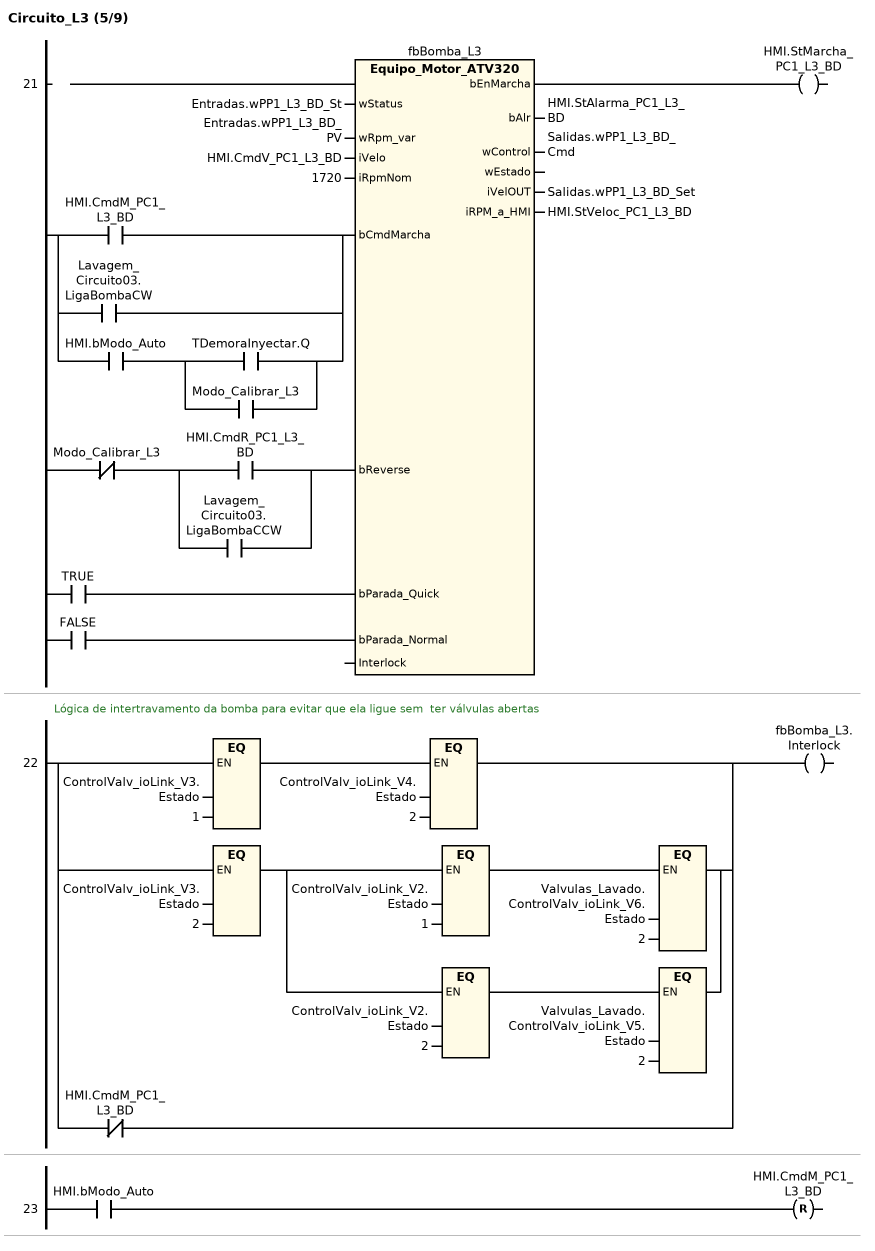
// NETWORK 21
fbBomba_L3(
    wStatus := Entradas.wPP1_L3_BD_St,
    wRpm_var := Entradas.wPP1_L3_BD_PV,
    iVelo := HMI.CmdV_PC1_L3_BD,
    iRpmNom := 1720,
    bCmdMarcha := HMI.CmdM_PC1_L3_BD OR Lavagem_Circuito03.LigaBombaCW OR HMI.bModo_Auto AND (TDemoraInyectar.Q OR Modo_Calibrar_L3),
    bReverse := NOT Modo_Calibrar_L3 AND (HMI.CmdR_PC1_L3_BD OR Lavagem_Circuito03.LigaBombaCCW),
    bParada_Quick := TRUE,
    bParada_Normal := FALSE,
    bAlr => HMI.StAlarma_PC1_L3_BD,
    wControl => Salidas.wPP1_L3_BD_Cmd,
    iVelOUT => Salidas.wPP1_L3_BD_Set,
    iRPM_a_HMI => HMI.StVeloc_PC1_L3_BD); // Equipo_Motor_ATV320
HMI.StMarcha_PC1_L3_BD := fbBomba_L3.bEnMarcha;

// NETWORK 22
// Lógica de intertravamento da bomba para evitar que ela ligue sem  ter válvulas abertas
_w6 := NOT HMI.CmdM_PC1_L3_BD;
IF NOT _w6 THEN
    _w7 := ControlValv_ioLink_V3.Estado = 2;
    _w6 := ControlValv_ioLink_V3.Estado = 1 AND ControlValv_ioLink_V4.Estado = 2 OR (_w7 AND ControlValv_ioLink_V2.Estado = 1 AND Valvulas_Lavado.ControlValv_ioLink_V6.Estado = 2 OR _w7 AND ControlValv_ioLink_V2.Estado = 2 AND Valvulas_Lavado.ControlValv_ioLink_V5.Estado = 2);
END_IF
fbBomba_L3.Interlock := _w6;

// NETWORK 23
HMI.CmdM_PC1_L3_BD R= HMI.bModo_Auto;

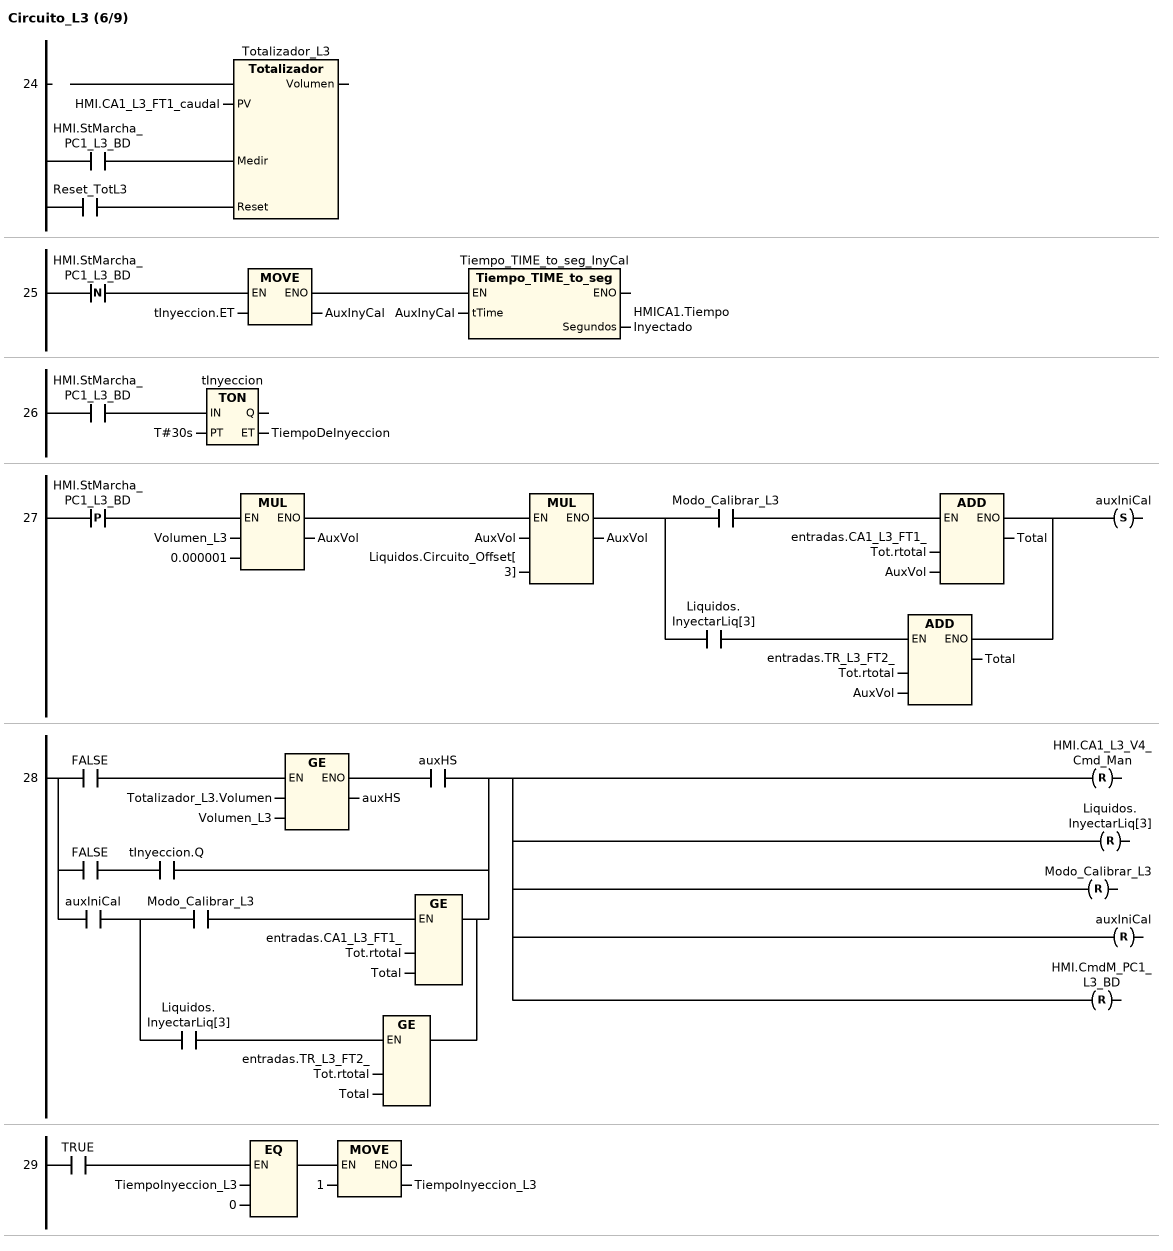
// NETWORK 24
Totalizador_L3(PV := HMI.CA1_L3_FT1_caudal, Medir := HMI.StMarcha_PC1_L3_BD, Reset := Reset_TotL3); // Totalizador

// NETWORK 25
_ft1(CLK := HMI.StMarcha_PC1_L3_BD);
_w8 := _ft1.Q;
IF _w8 THEN AuxInyCal := tInyeccion.ET; END_IF
IF _w8 THEN
    Tiempo_TIME_to_seg_InyCal(tTime := AuxInyCal, Segundos => HMICA1.TiempoInyectado); // Tiempo_TIME_to_seg
END_IF

// NETWORK 26
tInyeccion(IN := HMI.StMarcha_PC1_L3_BD, PT := T#30s, ET => TiempoDeInyeccion); // TON

// NETWORK 27
_rt1(CLK := HMI.StMarcha_PC1_L3_BD);
_w9 := _rt1.Q;
IF _w9 THEN AuxVol := Volumen_L3 * 0.000001; END_IF
IF _w9 THEN AuxVol := AuxVol * Liquidos.Circuito_Offset[3]; END_IF
IF _w9 AND Modo_Calibrar_L3 THEN Total := entradas.CA1_L3_FT1_Tot.rtotal + AuxVol; END_IF
IF _w9 AND Liquidos.InyectarLiq[3] THEN Total := entradas.TR_L3_FT2_Tot.rtotal + AuxVol; END_IF
auxIniCal S= _w9 AND Modo_Calibrar_L3 OR _w9 AND Liquidos.InyectarLiq[3];

// NETWORK 28
IF FALSE THEN auxHS := Totalizador_L3.Volumen >= Volumen_L3; END_IF
_w10 := FALSE AND auxHS OR FALSE AND tInyeccion.Q OR (auxIniCal AND Modo_Calibrar_L3 AND entradas.CA1_L3_FT1_Tot.rtotal >= Total OR auxIniCal AND Liquidos.InyectarLiq[3] AND entradas.TR_L3_FT2_Tot.rtotal >= Total);
HMI.CA1_L3_V4_Cmd_Man R= _w10;
Liquidos.InyectarLiq[3] R= _w10;
Modo_Calibrar_L3 R= _w10;
auxIniCal R= _w10;
HMI.CmdM_PC1_L3_BD R= _w10;

// NETWORK 29
IF TiempoInyeccion_L3 = 0 THEN TiempoInyeccion_L3 := 1; END_IF

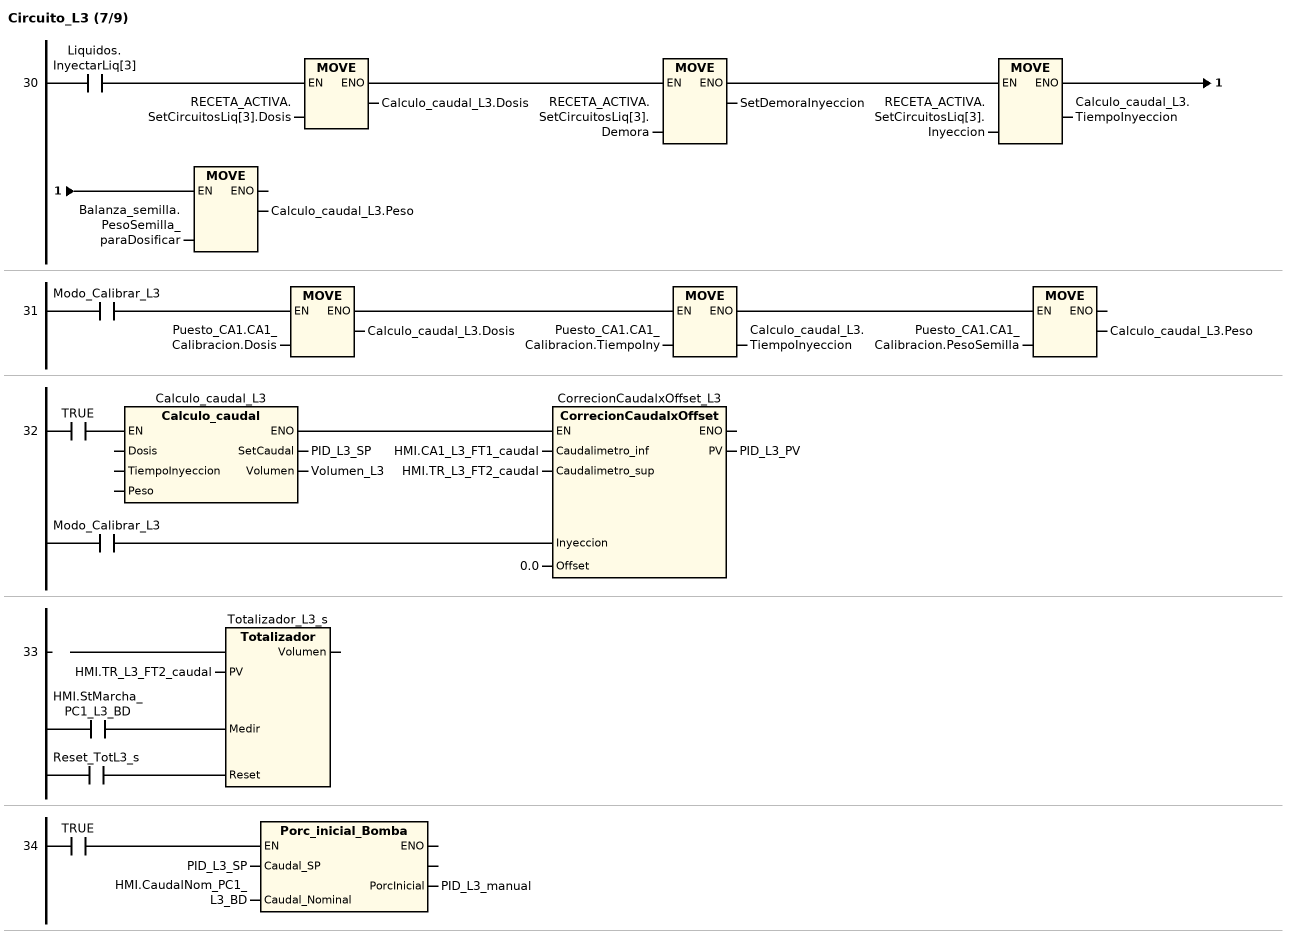
// NETWORK 30
_w11 := Liquidos.InyectarLiq[3];
IF _w11 THEN Calculo_caudal_L3.Dosis := RECETA_ACTIVA.SetCircuitosLiq[3].Dosis; END_IF
IF _w11 THEN SetDemoraInyeccion := RECETA_ACTIVA.SetCircuitosLiq[3].Demora; END_IF
IF _w11 THEN Calculo_caudal_L3.TiempoInyeccion := RECETA_ACTIVA.SetCircuitosLiq[3].Inyeccion; END_IF
IF _w11 THEN Calculo_caudal_L3.Peso := Balanza_semilla.PesoSemilla_paraDosificar; END_IF

// NETWORK 31
_w12 := Modo_Calibrar_L3;
IF _w12 THEN Calculo_caudal_L3.Dosis := Puesto_CA1.CA1_Calibracion.Dosis; END_IF
IF _w12 THEN Calculo_caudal_L3.TiempoInyeccion := Puesto_CA1.CA1_Calibracion.TiempoIny; END_IF
IF _w12 THEN Calculo_caudal_L3.Peso := Puesto_CA1.CA1_Calibracion.PesoSemilla; END_IF

// NETWORK 32
Calculo_caudal_L3(SetCaudal => PID_L3_SP, Volumen => Volumen_L3); // Calculo_caudal
CorrecionCaudalxOffset_L3(
    Caudalimetro_inf := HMI.CA1_L3_FT1_caudal,
    Caudalimetro_sup := HMI.TR_L3_FT2_caudal,
    Inyeccion := Modo_Calibrar_L3,
    Offset := 0.0,
    PV => PID_L3_PV); // CorrecionCaudalxOffset

// NETWORK 33
Totalizador_L3_s(PV := HMI.TR_L3_FT2_caudal, Medir := HMI.StMarcha_PC1_L3_BD, Reset := Reset_TotL3_s); // Totalizador

// NETWORK 34
Porc_inicial_Bomba(Caudal_SP := PID_L3_SP, Caudal_Nominal := HMI.CaudalNom_PC1_L3_BD, PorcInicial => PID_L3_manual);

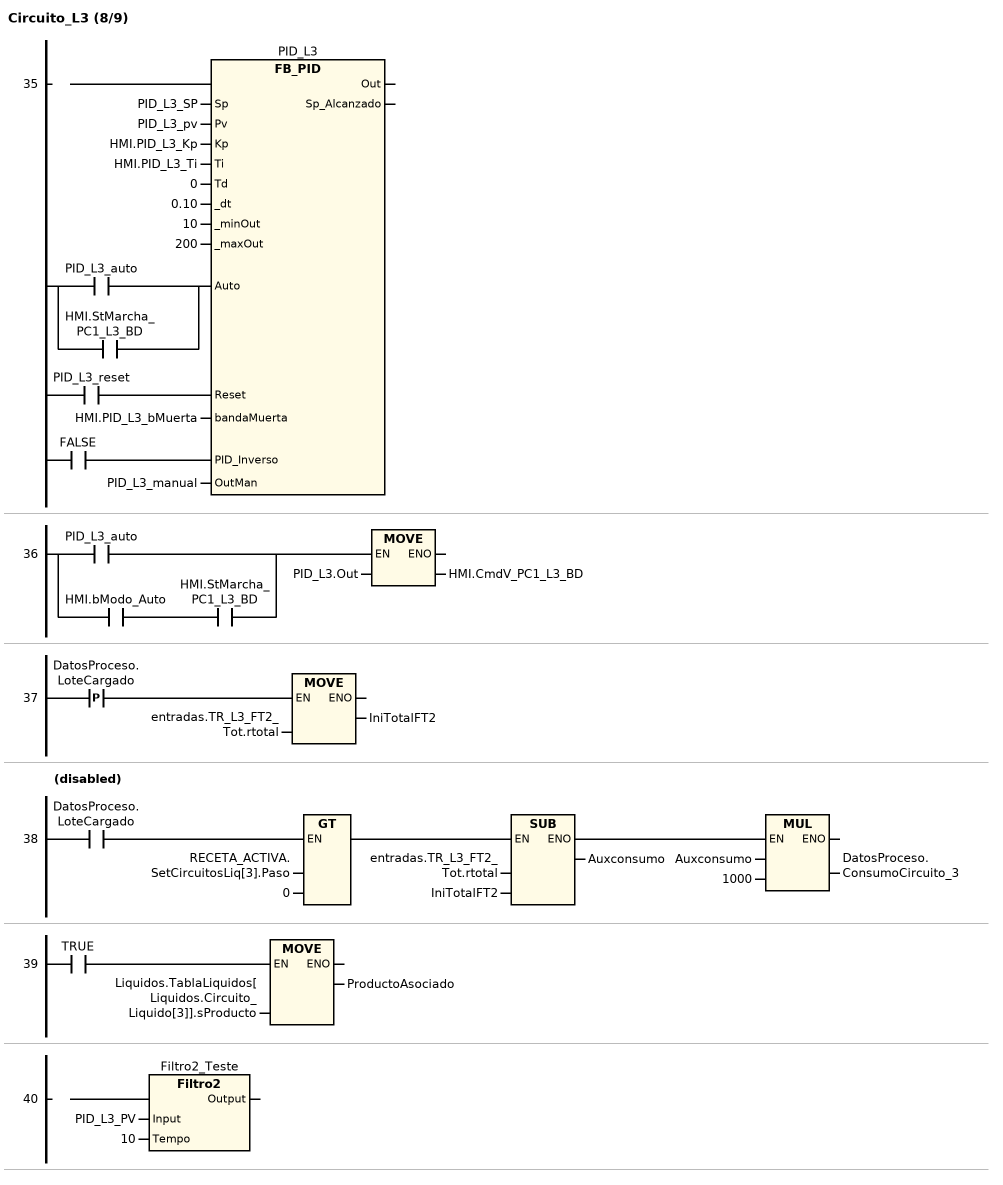
// NETWORK 35
PID_L3(
    Sp := PID_L3_SP,
    Pv := PID_L3_pv,
    Kp := HMI.PID_L3_Kp,
    Ti := HMI.PID_L3_Ti,
    Td := 0,
    _dt := 0.10,
    _minOut := 10,
    _maxOut := 200,
    Auto := PID_L3_auto OR HMI.StMarcha_PC1_L3_BD,
    Reset := PID_L3_reset,
    bandaMuerta := HMI.PID_L3_bMuerta,
    PID_Inverso := FALSE,
    OutMan := PID_L3_manual); // FB_PID

// NETWORK 36
IF PID_L3_auto OR HMI.bModo_Auto AND HMI.StMarcha_PC1_L3_BD THEN HMI.CmdV_PC1_L3_BD := PID_L3.Out; END_IF

// NETWORK 37
_rt2(CLK := DatosProceso.LoteCargado);
IF _rt2.Q THEN IniTotalFT2 := entradas.TR_L3_FT2_Tot.rtotal; END_IF

// NETWORK 38 (disabled)
// _w13 := DatosProceso.LoteCargado AND RECETA_ACTIVA.SetCircuitosLiq[3].Paso > 0;
// IF _w13 THEN Auxconsumo := entradas.TR_L3_FT2_Tot.rtotal - IniTotalFT2; END_IF
// IF _w13 THEN DatosProceso.ConsumoCircuito_3 := Auxconsumo * 1000; END_IF

// NETWORK 39
ProductoAsociado := Liquidos.TablaLiquidos[Liquidos.Circuito_Liquido[3]].sProducto;

// NETWORK 40
Filtro2_Teste(Input := PID_L3_PV, Tempo := 10); // Filtro2

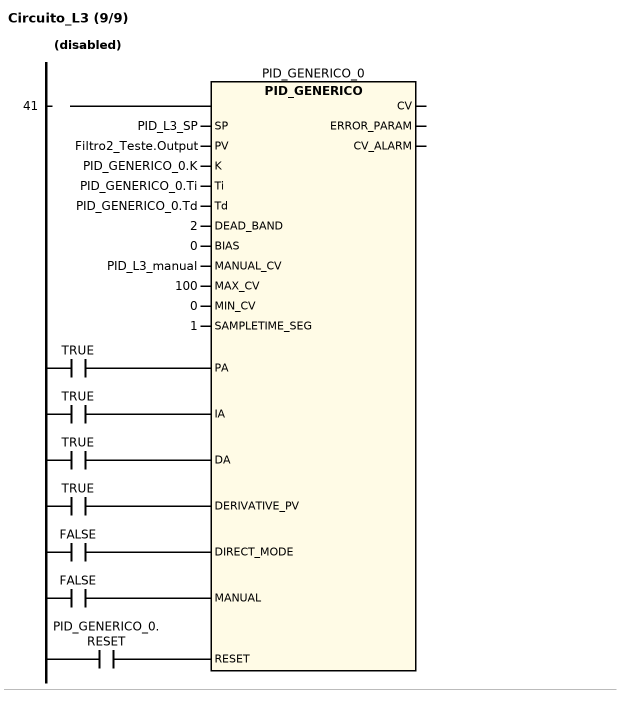
// NETWORK 41 (disabled)
// PID_GENERICO_0(
//     SP := PID_L3_SP,
//     PV := Filtro2_Teste.Output,
//     K := PID_GENERICO_0.K,
//     Ti := PID_GENERICO_0.Ti,
//     Td := PID_GENERICO_0.Td,
//     DEAD_BAND := 2,
//     BIAS := 0,
//     MANUAL_CV := PID_L3_manual,
//     MAX_CV := 100,
//     MIN_CV := 0,
//     SAMPLETIME_SEG := 1,
//     PA := TRUE,
//     IA := TRUE,
//     DA := TRUE,
//     DERIVATIVE_PV := TRUE,
//     DIRECT_MODE := FALSE,
//     MANUAL := FALSE,
//     RESET := PID_GENERICO_0.RESET); // PID_GENERICO

END_PROGRAM

// ---- POUs/TestesPID/PID_GENERICO.TcPOU
FUNCTION_BLOCK PID_GENERICO

VAR_INPUT
	SP: REAL; //SETPOINT
	PV: REAL; //VARIAVEL DE PROCESSO (ENTRADA)
	K: REAL; //GANHO PROPORCIONAL
	Ti: REAL; //GANHO INTEGRAL (TEMPO INTEGRAL)
	Td: REAL; //GANHO REAL (TEMPO DERIVATIVO)
	DEAD_BAND: REAL; //BANDA MORTA
	BIAS: REAL; //BIAS - VALOR SOMANDO A SAIDA DO CONTROLADOR
	MANUAL_CV: REAL; //VALOR DA SAIDA QUANDO O MANUAL ESTIVER HABILITADO
	MAX_CV: REAL; //VALOR MAXIMO DA SAIDA
	MIN_CV: REAL; //VALOR MINIMO DA SAIDA
	SAMPLETIME_SEG:REAL; //TEMPO DE ATUALIZAÇÃO DA TASK
	PA: BOOL; //HABILITA FATOR PROPORCIONAL
	IA: BOOL; //HABILITA FATOR INTEGRAL
	DA: BOOL; //HABILITA FATOR DERIVATIVO
	DERIVATIVE_PV: BOOL; //ADICIONAR FATOR DERIVATIVO A VARIAVEL DE PROCESSO
	DIRECT_MODE: BOOL; //MODO DIRETO OU REVERSO
	MANUAL: BOOL; //HABILITA MODO MANUAL
	RESET: BOOL; //RESET DO BLOCO
END_VAR
VAR_OUTPUT
	CV: INT; //VARIAVEL DE CONTROLE (SAIDA)
	ERROR_PARAM: BOOL; //ERRO DE PARAMETRO
	CV_ALARM: BOOL; //ALARME DE LIMITES DA SAIDA ATINGIDO (SATURAÇÃO)
END_VAR
VAR
	RealCV : REAL := 0;
	RealTimeCycle: ARRAY [0..2] OF REAL := [0,0,0];
	RealSystemError: ARRAY [0..3] OF REAL := [0,0,0,0];
	RealProcessVariable: ARRAY [0..3] OF REAL := [0,0,0,0];
	RealProportionalAction: REAL := 0;
	RealIntegralAction: REAL := 0;
	RealDerivativeAction: REAL := 0;
	RealIntegralLastAction: REAL := 0;
	DwCurrentReferenceCycle: DWORD;
	DwLastReferenceCycle:DWORD := 0;
	BoolFirstCycle: BOOL := TRUE;
END_VAR


(*###################################################################################                                                     
##  									                                      								                                      
##	Function Block Name: PID_FB                                                                                                                                  
##  									                                      								                                      
##  Version: 1.00                                                                                                                                                                 
##  									                                      								                                      
##                                                                                                
##  									                                      								                                      
##  Software Description: The PID function block implements the proportional, integral and derivative          
##  control algorithm. Using a process variable (PV) and a setpoint (SP) the function computes the              
##  control variable (CV) for the process under control. This value is calculated periodically, and 
##  takes into consideration the proportional, integral and derivative configured factors. This is a ISA 
##  PID control algorithm in which the proportional gain is the controller gain, that is applied to the 
##  controller error as well as it's integral and derivative terms.
##
###################################################################################*)




(* ----------------------------------------------------------  RESET TREATMENT-------------------------------------------------------*)
IF(RESET = TRUE)
THEN
		RealSystemError[0] := 0;
		RealSystemError[1] := 0;
		RealSystemError[2] := 0;
		RealSystemError[3] := 0;
		RealProcessVariable[0] := 0;
		RealProcessVariable[1] := 0;
		RealProcessVariable[2] := 0;
		RealProcessVariable[3] := 0;
		RealTimeCycle[0] := 0;
		RealTimeCycle[1] := 0;
		RealTimeCycle[2] := 0;
		RealIntegralLastAction := 0;
		BoolFirstCycle:= TRUE;

		(* Reset the output variables*)
		ERROR_PARAM := FALSE;
		CV_ALARM := FALSE;
		CV := 0;
		RETURN;
END_IF;
(*############################## END OF RESET TREATMENT ############################*)


(*------------------------------------------------------- PARAMETERS TEST -----------------------------------------------------------*)
IF(K<=0 OR Ti<=0 OR Td<0 OR MAX_CV<MIN_CV OR MAX_CV>32767 OR MIN_CV<-32768)
THEN
		RealSystemError[0] := 0;
		RealSystemError[1] := 0;
		RealSystemError[2] := 0;
		RealSystemError[3] := 0;
		RealProcessVariable[0] := 0;
		RealProcessVariable[1] := 0;
		RealProcessVariable[2] := 0;
		RealProcessVariable[3] := 0;
		RealTimeCycle[0] := 0;
		RealTimeCycle[1] := 0;
		RealTimeCycle[2] := 0;
		RealIntegralLastAction := 0;
		BoolFirstCycle:= TRUE;
		CV_ALARM := FALSE;
		ERROR_PARAM:= TRUE;
		CV:= 0;
		RETURN;
ELSE
		ERROR_PARAM:= FALSE;
END_IF;

(*############################## END PARAMETERS TEST ###############################*)

(*------------------ KEEPS A LOG OF THE LAST FOUR ERRORS  AND PROCESS VARIABLES ----------------------*)

RealSystemError[3] := RealSystemError[2];
RealSystemError[2] := RealSystemError[1];
RealSystemError[1] := RealSystemError[0];

RealProcessVariable[3] := RealProcessVariable[2];
RealProcessVariable[2] := RealProcessVariable[1];
RealProcessVariable[1] := RealProcessVariable[0];

IF(DIRECT_MODE = TRUE)
THEN	RealSystemError[0]:=PV - SP;
		RealProcessVariable[0 ]:= -PV;

ELSE	RealSystemError[0]:=SP -PV;
		RealProcessVariable[0 ]:= PV;
END_IF;


(*  Applys the dead band over the system error *)
IF(ABS(RealSystemError[0]) <= ABS(DEAD_BAND))
THEN	RealSystemError[0]:= 0;
END_IF;

(*################################ END OF ERRORS AND PV LOG ############################*)


(*------------------------------------------------------ TIME BASE DEFINITION ----------------------------------------------------------*)


IF(BoolFirstCycle = FALSE)
THEN
		RealTimeCycle[2] := SAMPLETIME_SEG;
		RealTimeCycle[1] := SAMPLETIME_SEG;
		RealTimeCycle[0]:= SAMPLETIME_SEG;

		IF(RealTimeCycle[0] = 0)		(* If the current cycle is less than 1 ms it is forced do 1 ms *)
		THEN	RealTimeCycle[0] := 0.001;
		END_IF;
ELSE
		BoolFirstCycle := FALSE;
		RETURN;
END_IF;
(*############################# END OF TIME BASE DEFINITION  ############################*)


(* -----------------------------------------------------  PROPORTIONAL ACTION -----------------------------------------------------*)
 IF (PA = TRUE)
THEN
		(* The proportional action is only the current error *)
		(* Remind that "K" is the controller gain and it will be applied to the sum of proportional integral and derivative actions *)
		RealProportionalAction := RealSystemError[0];
ELSE
		(* If the proportional action is not desirable its value would be zero *)
		RealProportionalAction := 0;
END_IF;
(*############################ END OF PROPORTIONAL ACTION #############################*)


(* ---------------------------------------------------------  INTEGRAL ACTION ---------------------------------------------------------*)
IF( IA = TRUE AND MANUAL = FALSE)
THEN
		(* It keeps the last egral Action because it must be used when the controled variable reaches its limits *)
		RealIntegralLastAction := RealIntegralAction;

		(* The integral action is the amount  obtained from the current system error multiplied by the sample time and
		    divided by  the the programmed integral time*)

		(* Remind that "K" is the controller gain and it will be applied to the sum of proportional integral and derivative actions *)
		RealIntegralAction := RealIntegralLastAction + RealSystemError[0] * RealTimeCycle[0] / Ti;

		(* Limits the integral action in 10 times the maximum output *)
		IF(RealIntegralAction > 327670)
		THEN	RealIntegralAction := 327670;
		END_IF;

		IF(RealIntegralAction < -327670)
		THEN	RealIntegralAction := -327670;
		END_IF;
ELSE
		(* If the Integral action is not desirable its value will be zero *)
		RealIntegralAction:= 0;
END_IF;
(*################################ END OF INTEGRAL ACTION ##############################*)


(* --------------------------------------------------------  DERIVATIVE ACTION --------------------------------------------------------*)
IF (DA = TRUE)
THEN
		(* The derivative action is the variation of de error during 3 cycles multiplied by the programmed derivative time*)
		(* Remind that "K" is the controller gain and it will be applied to the sum of proportional integral and derivative actions *)
		IF(DERIVATIVE_PV = TRUE)
		THEN	RealDerivativeAction:=  Td * (RealProcessVariable[3] - RealProcessVariable[0]) / (RealTimeCycle[0] + RealTimeCycle[1] + RealTimeCycle[2]);
		ELSE	RealDerivativeAction:=  Td * (RealSystemError[0] - RealSystemError[3]) / (RealTimeCycle[0] + RealTimeCycle[1] + RealTimeCycle[2]);
		END_IF;

		(* Limits the derivative action in 10 times the maximum output *)
		IF(RealDerivativeAction > 327670)
		THEN	RealDerivativeAction := 327670;
		END_IF;

		IF(RealDerivativeAction < -327670)
		THEN	RealDerivativeAction := -327670;
		END_IF;
ELSE
		(* If the derivative action is not desirable its value will be zero *)
		RealDerivativeAction:=0;
END_IF;
(*###############################  END OF DERIVATIVE ACTION ############################*)


(*-------------------------------------------- TESTS MANUAL OR AUTOMATIC MODE -----------------------------------------*)
IF(MANUAL = FALSE)
THEN
		(* in automatic mode the control variable is the sum of  the three actions  *)
		RealCV := K*(RealProportionalAction + RealIntegralAction + RealDerivativeAction) + BIAS;

		(* limits the output in the maximum programmed *)
		IF(RealCV > MAX_CV)
		THEN	CV := REAL_TO_INT(MAX_CV);
				CV_ALARM := TRUE;    (*indicates that the ouput reaches the limit*)
				(* keeps the current Integral Action only if the system error is negative *)
				IF(RealSystemError[0] > 0)
				THEN	RealIntegralAction := RealIntegralLastAction;
				END_IF;

		(* limits the output in the minimum programmed *)
		ELSE	IF(RealCV <  MIN_CV)
				THEN	CV := REAL_TO_INT(MIN_CV);
						CV_ALARM := TRUE;     (*indicates that the ouput reaches the limit*)
						(* keeps the current Integral Action only if the system error is positive *)
						IF(RealSystemError[0] < 0)
						THEN	RealIntegralAction := RealIntegralLastAction;
						END_IF;
				ELSE	CV := REAL_TO_INT(RealCV);
						CV_ALARM := FALSE;    (*indicates that the ouput is between the limits*)
				END_IF;
		END_IF;
ELSE
		(*In  manual mode the manual value is copied to the control variable .
		The stored integral action will be the difference between the CV_MANUAL and the Proportional, Derivative Actions
		and the programmed FF_Bias. *)

		(* If the Manual CV is configured above or below to the limits the control variable alarm is set and the CV will be
                 forced to the closest limit*)

		IF(MANUAL_CV > MAX_CV)
		THEN	CV := REAL_TO_INT(MAX_CV);
				CV_ALARM := TRUE;
		ELSE
				IF(MANUAL_CV <MIN_CV)
			    	THEN	CV := REAL_TO_INT(MIN_CV);
						CV_ALARM := TRUE;

				ELSE	CV := REAL_TO_INT(MANUAL_CV);
						CV_ALARM := FALSE;

				END_IF;
		END_IF;

		(*This Integral Action will be used in case of switch to automatic mode to ensure a smooth transition. *)
		RealIntegralAction:= (INT_TO_REAL(CV) - BIAS) / K - RealProportionalAction - RealDerivativeAction;

END_IF;

(*###############################  END MANUAL / AUTOMATIC ############################*)

END_FUNCTION_BLOCK

// ---- POUs/Secuencias/Porc_inicial_Bomba.TcPOU
FUNCTION Porc_inicial_Bomba : BOOL
VAR_INPUT
	Caudal_SP:REAL;
	Caudal_Nominal:REAL;
END_VAR
VAR_OUTPUT
	PorcInicial:REAL;
END_VAR
VAR
END_VAR

IF Caudal_Nominal=0 THEN
	Caudal_Nominal:=1;
END_IF
PorcInicial:=(Caudal_SP/Caudal_Nominal)*100.0*1.0;

END_FUNCTION

// ---- POUs/Puesto_Calibracion_1/Circuito_L4.TcPOU
PROGRAM Circuito_L4
VAR_INPUT
	Modo_Calibrar_L4: BOOL;
END_VAR
	
VAR
		fbBomba_L4 :Equipo_Motor_ATV320;
		ControlValv_ioLink_V1:ControlValv_ioLink;
		ControlValv_ioLink_V2: ControlValv_ioLink;
		ControlValv_ioLink_V3: ControlValv_ioLink;
		ControlValv_ioLink_V4: ControlValv_ioLink;
		Falla_L4_V1:BOOL;
		Falla_L4_V2:BOOL;
		Falla_L4_V3:BOOL;
		Falla_L4_V4:BOOL;
	Balanza_PU1_WT4: Balanza;
		dHS:DINT;
		TOF_calibradoIBC: TOF;
		TDemoraInyectar: TON;
		SetDemoraInyeccion: REAL;
	

	Volumen_L4: REAL;
	AuxVol: REAL;
	Total: REAL;
	auxIniCal: BOOL;
	Calculo_caudal_L4: Calculo_caudal;
	PID_L4_SP: REAL;
	PID_L4_PV: REAL;
	CorrecionCaudalxOffset_L4: CorrecionCaudalxOffset;
	tInyeccion: TON;
	PID_L4_manual: REAL;
	PID_L4: FB_PID;
	PID_L4_Kp: REAL := 0.1;
	PID_L4_Ti: REAL := 100;
	PID_L4_auto: BOOL;
	PID_L4_reset: BOOL;
	PID_L4_bMuerta: REAL := 5;
	Tiempo_seg_to_TIME_DemoraInyec: Tiempo_seg_to_TIME;
	AuxTDemoraInyec: TIME;
	Tiempo_TIME_to_seg_InyCal: Tiempo_TIME_to_seg;
	AuxInyCal:TIME;
	IniTotalFT2:REAL;
	Auxconsumo:REAL;
	ProductoAsociado: STRING;
	Lavagem_Circuito04: Lavagem;
	
END_VAR
VAR PERSISTENT
	UltimaCalibracao	:UDINT;	//Data e hora da ultima calibração
END_VAR
VAR // added by the converter: edge detectors and wires of the graphical bodies
    _w1, _w2, _w3, _w4, _w5, _w6, _w7, _w8, _w9, _w10, _w11, _w12, _w13 : BOOL;
    _ft1 : F_TRIG;
    _rt1, _rt2 : R_TRIG;
END_VAR

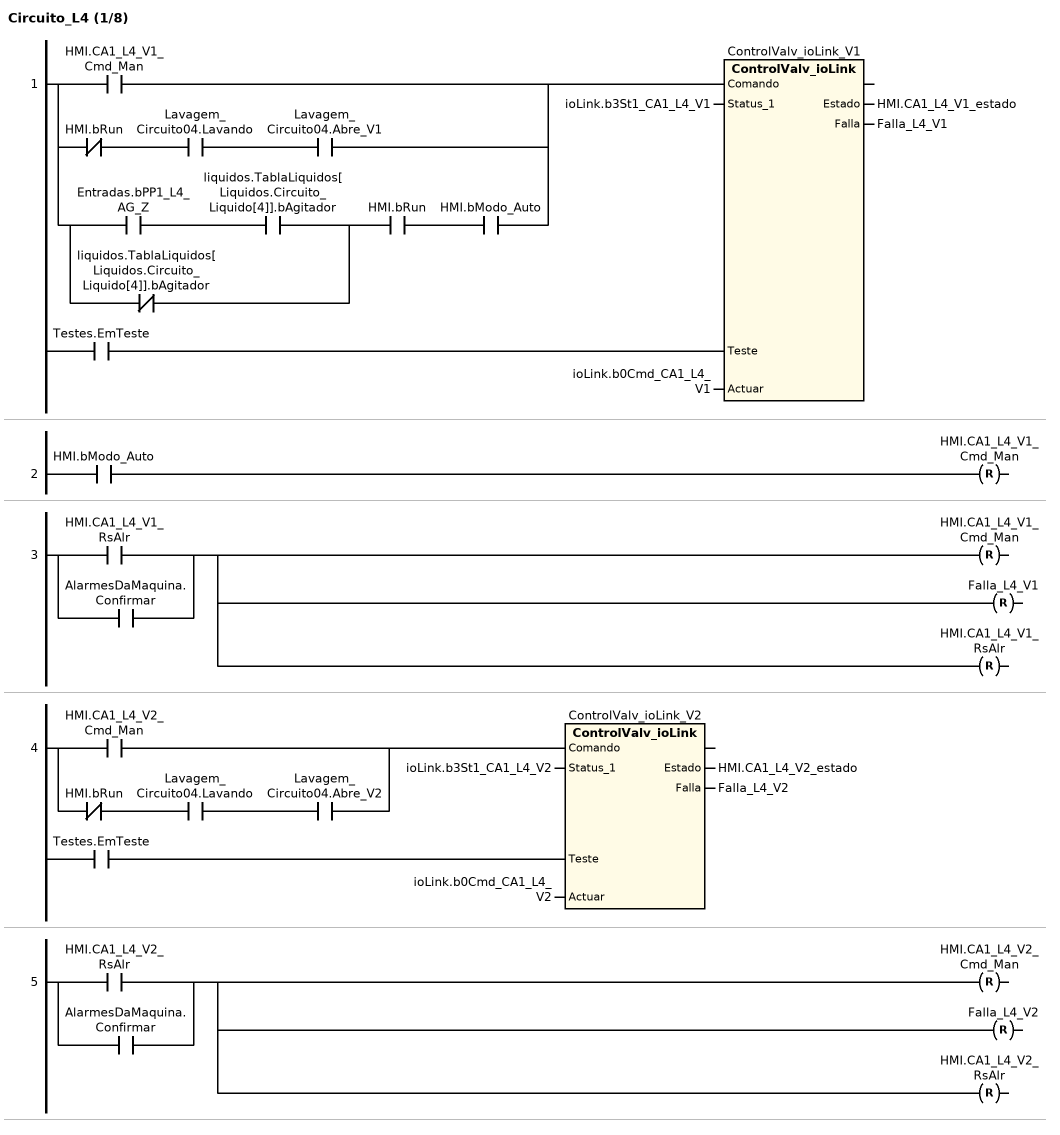
// NETWORK 1
ControlValv_ioLink_V1(
    Comando := HMI.CA1_L4_V1_Cmd_Man OR NOT HMI.bRun AND Lavagem_Circuito04.Lavando AND Lavagem_Circuito04.Abre_V1 OR (Entradas.bPP1_L4_AG_Z AND (liquidos.TablaLiquidos[Liquidos.Circuito_Liquido[4]].bAgitador) OR NOT (liquidos.TablaLiquidos[Liquidos.Circuito_Liquido[4]].bAgitador)) AND HMI.bRun AND HMI.bModo_Auto,
    Status_1 := ioLink.b3St1_CA1_L4_V1,
    Teste := Testes.EmTeste,
    Actuar := ioLink.b0Cmd_CA1_L4_V1,
    Estado => HMI.CA1_L4_V1_estado,
    Falla => Falla_L4_V1); // ControlValv_ioLink

// NETWORK 2
HMI.CA1_L4_V1_Cmd_Man R= HMI.bModo_Auto;

// NETWORK 3
_w1 := HMI.CA1_L4_V1_RsAlr OR AlarmesDaMaquina.Confirmar;
HMI.CA1_L4_V1_Cmd_Man R= _w1;
Falla_L4_V1 R= _w1;
HMI.CA1_L4_V1_RsAlr R= _w1;

// NETWORK 4
ControlValv_ioLink_V2(
    Comando := HMI.CA1_L4_V2_Cmd_Man OR NOT HMI.bRun AND Lavagem_Circuito04.Lavando AND Lavagem_Circuito04.Abre_V2,
    Status_1 := ioLink.b3St1_CA1_L4_V2,
    Teste := Testes.EmTeste,
    Actuar := ioLink.b0Cmd_CA1_L4_V2,
    Estado => HMI.CA1_L4_V2_estado,
    Falla => Falla_L4_V2); // ControlValv_ioLink

// NETWORK 5
_w2 := HMI.CA1_L4_V2_RsAlr OR AlarmesDaMaquina.Confirmar;
HMI.CA1_L4_V2_Cmd_Man R= _w2;
Falla_L4_V2 R= _w2;
HMI.CA1_L4_V2_RsAlr R= _w2;

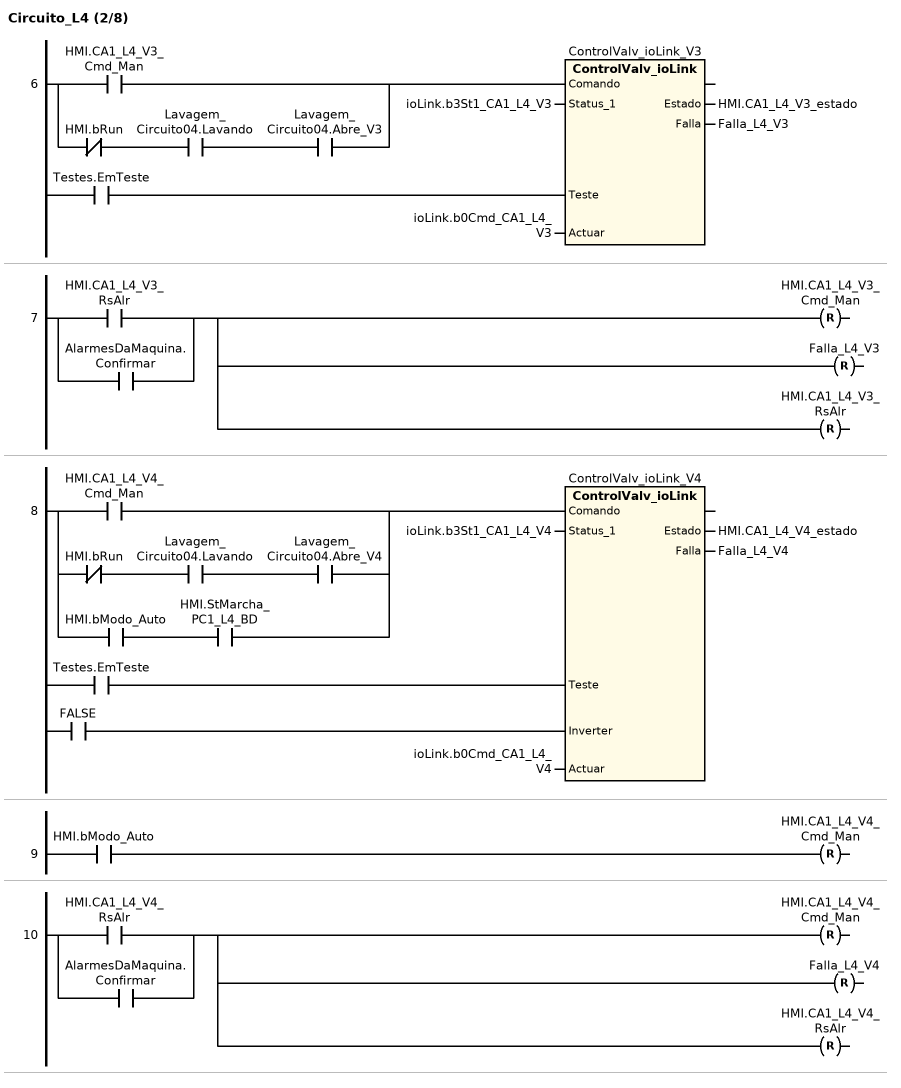
// NETWORK 6
ControlValv_ioLink_V3(
    Comando := HMI.CA1_L4_V3_Cmd_Man OR NOT HMI.bRun AND Lavagem_Circuito04.Lavando AND Lavagem_Circuito04.Abre_V3,
    Status_1 := ioLink.b3St1_CA1_L4_V3,
    Teste := Testes.EmTeste,
    Actuar := ioLink.b0Cmd_CA1_L4_V3,
    Estado => HMI.CA1_L4_V3_estado,
    Falla => Falla_L4_V3); // ControlValv_ioLink

// NETWORK 7
_w3 := HMI.CA1_L4_V3_RsAlr OR AlarmesDaMaquina.Confirmar;
HMI.CA1_L4_V3_Cmd_Man R= _w3;
Falla_L4_V3 R= _w3;
HMI.CA1_L4_V3_RsAlr R= _w3;

// NETWORK 8
ControlValv_ioLink_V4(
    Comando := HMI.CA1_L4_V4_Cmd_Man OR NOT HMI.bRun AND Lavagem_Circuito04.Lavando AND Lavagem_Circuito04.Abre_V4 OR HMI.bModo_Auto AND HMI.StMarcha_PC1_L4_BD,
    Status_1 := ioLink.b3St1_CA1_L4_V4,
    Teste := Testes.EmTeste,
    Inverter := FALSE,
    Actuar := ioLink.b0Cmd_CA1_L4_V4,
    Estado => HMI.CA1_L4_V4_estado,
    Falla => Falla_L4_V4); // ControlValv_ioLink

// NETWORK 9
HMI.CA1_L4_V4_Cmd_Man R= HMI.bModo_Auto;

// NETWORK 10
_w4 := HMI.CA1_L4_V4_RsAlr OR AlarmesDaMaquina.Confirmar;
HMI.CA1_L4_V4_Cmd_Man R= _w4;
Falla_L4_V4 R= _w4;
HMI.CA1_L4_V4_RsAlr R= _w4;

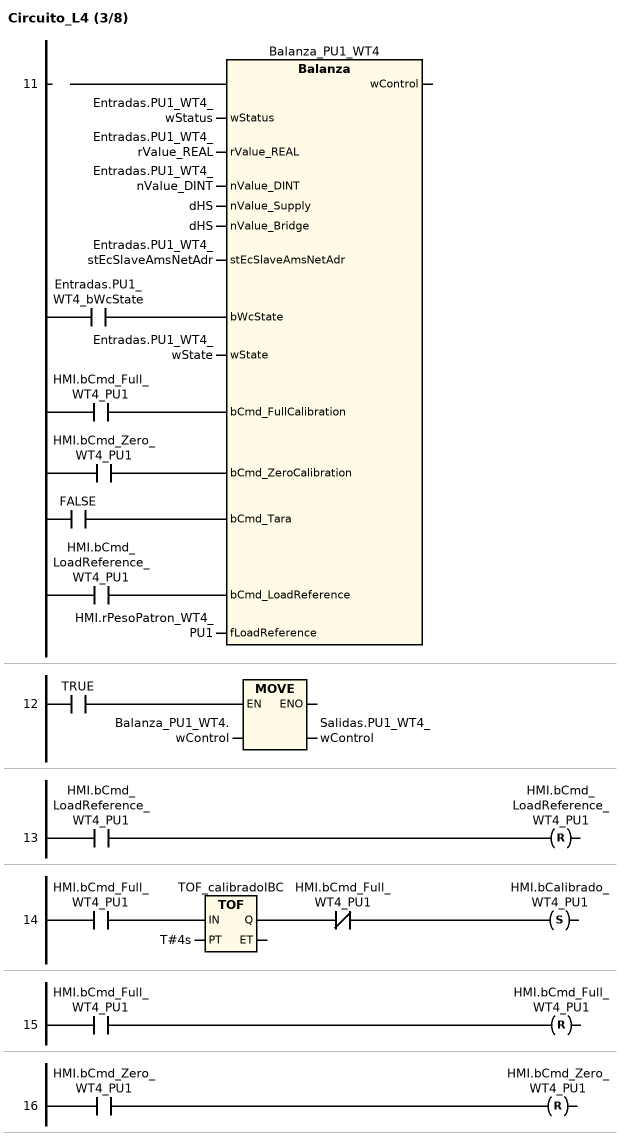
// NETWORK 11
Balanza_PU1_WT4(
    wStatus := Entradas.PU1_WT4_wStatus,
    rValue_REAL := Entradas.PU1_WT4_rValue_REAL,
    nValue_DINT := Entradas.PU1_WT4_nValue_DINT,
    nValue_Supply := dHS,
    nValue_Bridge := dHS,
    stEcSlaveAmsNetAdr := Entradas.PU1_WT4_stEcSlaveAmsNetAdr,
    bWcState := Entradas.PU1_WT4_bWcState,
    wState := Entradas.PU1_WT4_wState,
    bCmd_FullCalibration := HMI.bCmd_Full_WT4_PU1,
    bCmd_ZeroCalibration := HMI.bCmd_Zero_WT4_PU1,
    bCmd_Tara := FALSE,
    bCmd_LoadReference := HMI.bCmd_LoadReference_WT4_PU1,
    fLoadReference := HMI.rPesoPatron_WT4_PU1); // Balanza

// NETWORK 12
Salidas.PU1_WT4_wControl := Balanza_PU1_WT4.wControl;

// NETWORK 13
HMI.bCmd_LoadReference_WT4_PU1 R= HMI.bCmd_LoadReference_WT4_PU1;

// NETWORK 14
TOF_calibradoIBC(IN := HMI.bCmd_Full_WT4_PU1, PT := T#4s); // TOF
HMI.bCalibrado_WT4_PU1 S= TOF_calibradoIBC.Q AND NOT HMI.bCmd_Full_WT4_PU1;

// NETWORK 15
HMI.bCmd_Full_WT4_PU1 R= HMI.bCmd_Full_WT4_PU1;

// NETWORK 16
HMI.bCmd_Zero_WT4_PU1 R= HMI.bCmd_Zero_WT4_PU1;

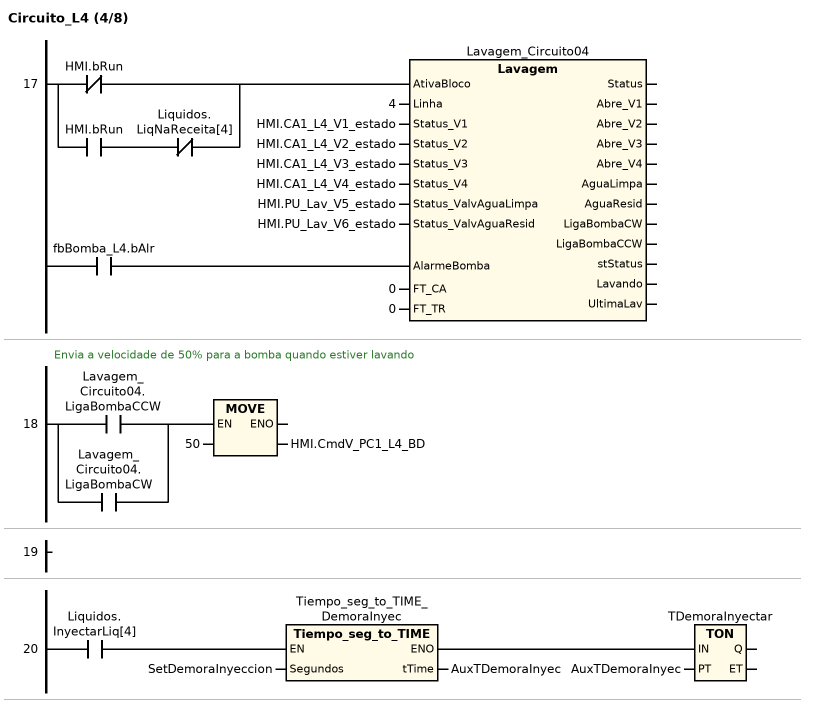
// NETWORK 17
Lavagem_Circuito04(
    AtivaBloco := NOT HMI.bRun OR HMI.bRun AND NOT Liquidos.LiqNaReceita[4],
    Linha := 4,
    Status_V1 := HMI.CA1_L4_V1_estado,
    Status_V2 := HMI.CA1_L4_V2_estado,
    Status_V3 := HMI.CA1_L4_V3_estado,
    Status_V4 := HMI.CA1_L4_V4_estado,
    Status_ValvAguaLimpa := HMI.PU_Lav_V5_estado,
    Status_ValvAguaResid := HMI.PU_Lav_V6_estado,
    AlarmeBomba := fbBomba_L4.bAlr,
    FT_CA := 0,
    FT_TR := 0); // Lavagem

// NETWORK 18
// Envia a velocidade de 50% para a bomba quando estiver lavando
IF Lavagem_Circuito04.LigaBombaCCW OR Lavagem_Circuito04.LigaBombaCW THEN HMI.CmdV_PC1_L4_BD := 50; END_IF

// NETWORK 19

// NETWORK 20
_w5 := Liquidos.InyectarLiq[4];
IF _w5 THEN
    Tiempo_seg_to_TIME_DemoraInyec(Segundos := SetDemoraInyeccion, tTime => AuxTDemoraInyec); // Tiempo_seg_to_TIME
END_IF
TDemoraInyectar(IN := _w5, PT := AuxTDemoraInyec); // TON

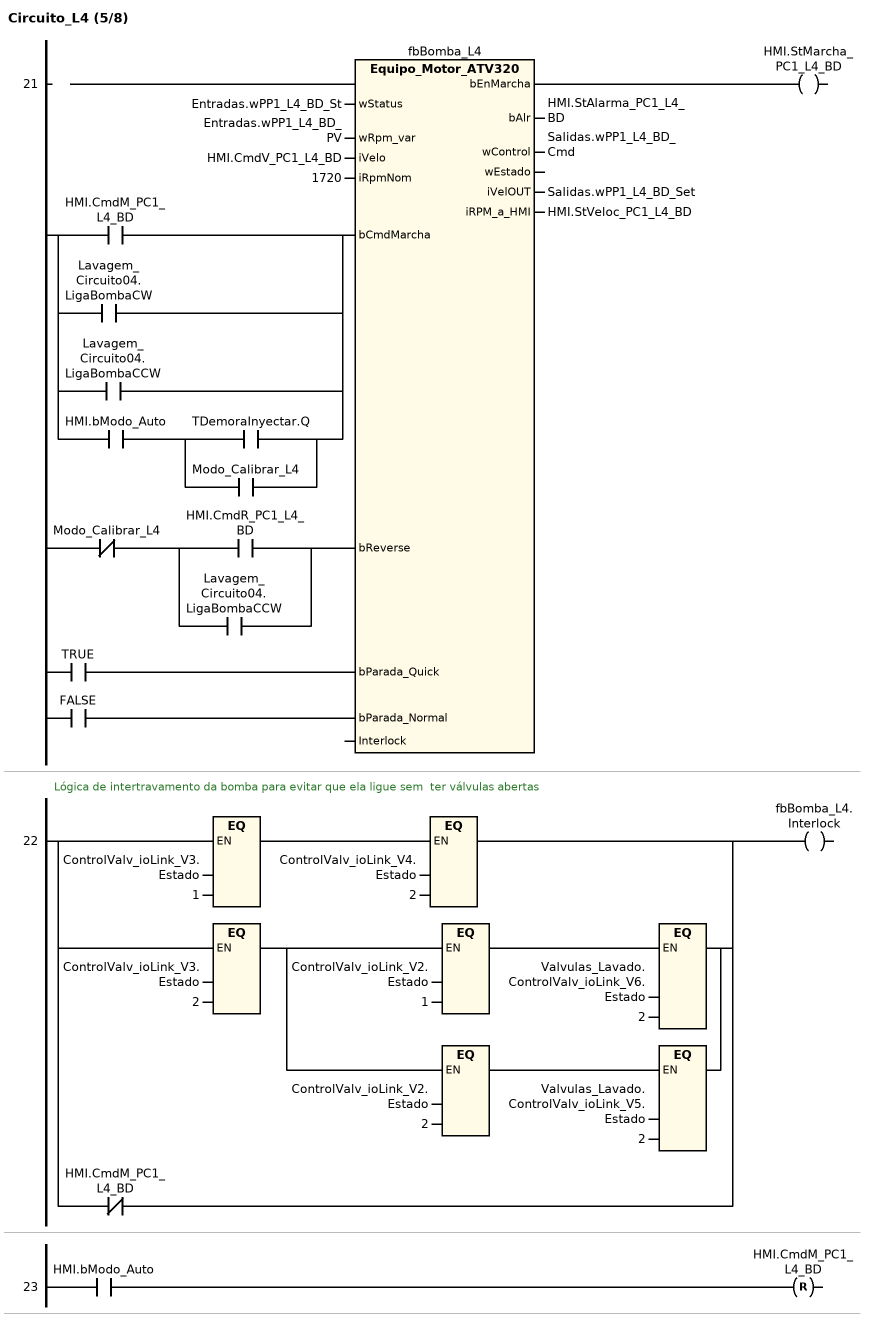
// NETWORK 21
fbBomba_L4(
    wStatus := Entradas.wPP1_L4_BD_St,
    wRpm_var := Entradas.wPP1_L4_BD_PV,
    iVelo := HMI.CmdV_PC1_L4_BD,
    iRpmNom := 1720,
    bCmdMarcha := HMI.CmdM_PC1_L4_BD OR Lavagem_Circuito04.LigaBombaCW OR Lavagem_Circuito04.LigaBombaCCW OR HMI.bModo_Auto AND (TDemoraInyectar.Q OR Modo_Calibrar_L4),
    bReverse := NOT Modo_Calibrar_L4 AND (HMI.CmdR_PC1_L4_BD OR Lavagem_Circuito04.LigaBombaCCW),
    bParada_Quick := TRUE,
    bParada_Normal := FALSE,
    bAlr => HMI.StAlarma_PC1_L4_BD,
    wControl => Salidas.wPP1_L4_BD_Cmd,
    iVelOUT => Salidas.wPP1_L4_BD_Set,
    iRPM_a_HMI => HMI.StVeloc_PC1_L4_BD); // Equipo_Motor_ATV320
HMI.StMarcha_PC1_L4_BD := fbBomba_L4.bEnMarcha;

// NETWORK 22
// Lógica de intertravamento da bomba para evitar que ela ligue sem  ter válvulas abertas
_w6 := NOT HMI.CmdM_PC1_L4_BD;
IF NOT _w6 THEN
    _w7 := ControlValv_ioLink_V3.Estado = 2;
    _w6 := ControlValv_ioLink_V3.Estado = 1 AND ControlValv_ioLink_V4.Estado = 2 OR (_w7 AND ControlValv_ioLink_V2.Estado = 1 AND Valvulas_Lavado.ControlValv_ioLink_V6.Estado = 2 OR _w7 AND ControlValv_ioLink_V2.Estado = 2 AND Valvulas_Lavado.ControlValv_ioLink_V5.Estado = 2);
END_IF
fbBomba_L4.Interlock := _w6;

// NETWORK 23
HMI.CmdM_PC1_L4_BD R= HMI.bModo_Auto;

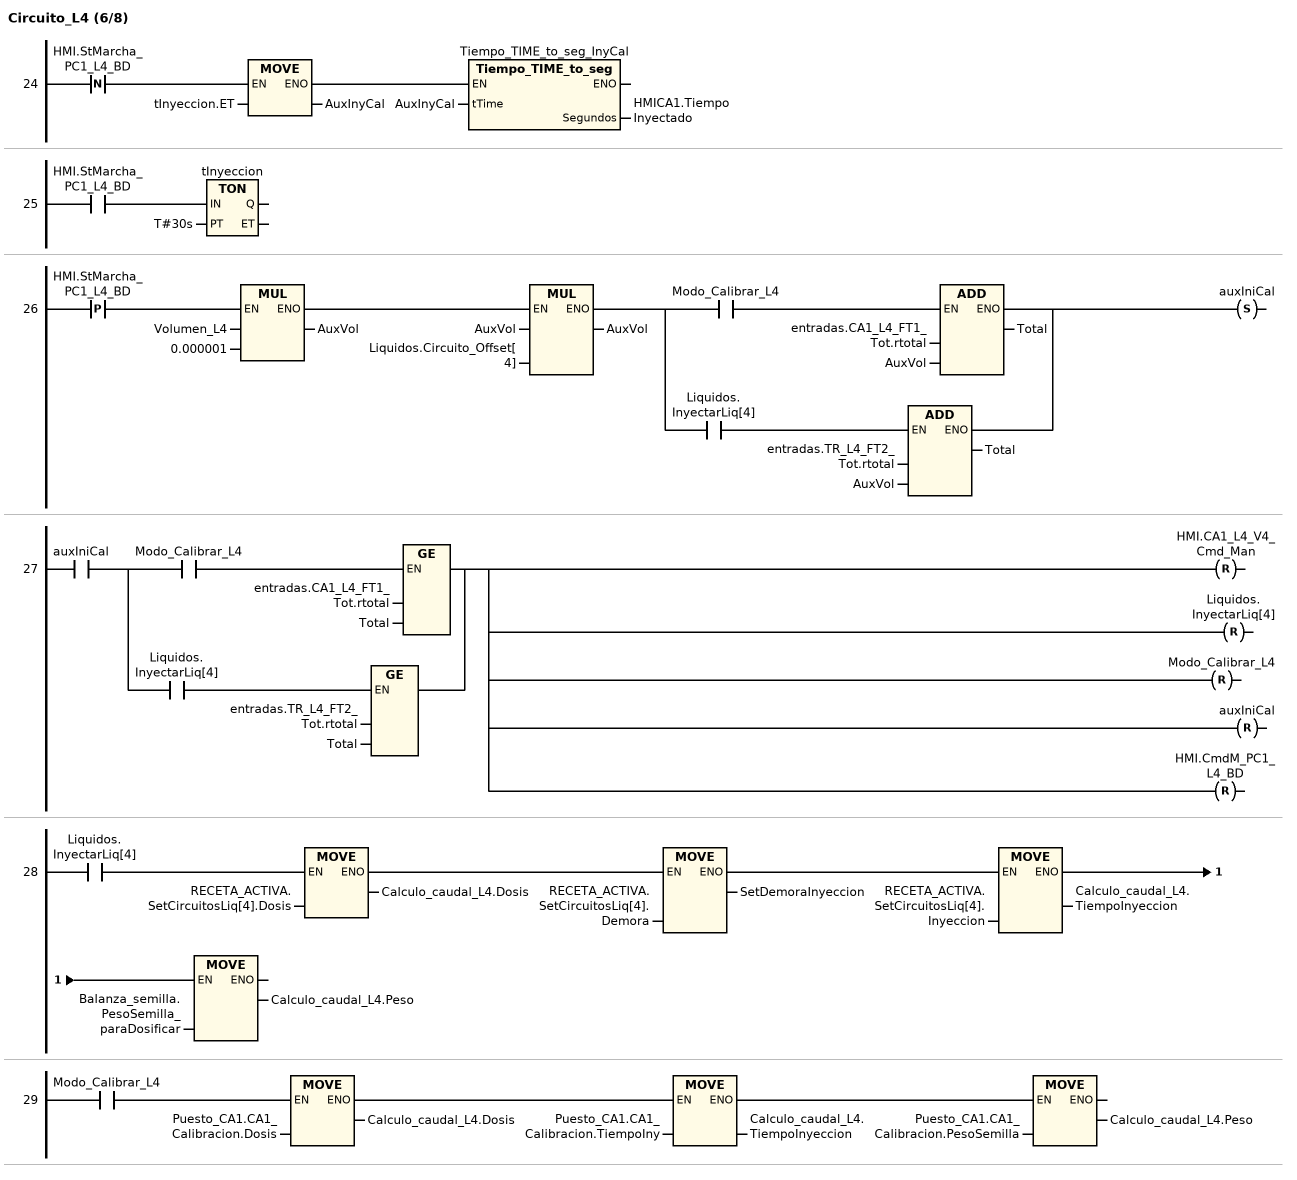
// NETWORK 24
_ft1(CLK := HMI.StMarcha_PC1_L4_BD);
_w8 := _ft1.Q;
IF _w8 THEN AuxInyCal := tInyeccion.ET; END_IF
IF _w8 THEN
    Tiempo_TIME_to_seg_InyCal(tTime := AuxInyCal, Segundos => HMICA1.TiempoInyectado); // Tiempo_TIME_to_seg
END_IF

// NETWORK 25
tInyeccion(IN := HMI.StMarcha_PC1_L4_BD, PT := T#30s); // TON

// NETWORK 26
_rt1(CLK := HMI.StMarcha_PC1_L4_BD);
_w9 := _rt1.Q;
IF _w9 THEN AuxVol := Volumen_L4 * 0.000001; END_IF
IF _w9 THEN AuxVol := AuxVol * Liquidos.Circuito_Offset[4]; END_IF
IF _w9 AND Modo_Calibrar_L4 THEN Total := entradas.CA1_L4_FT1_Tot.rtotal + AuxVol; END_IF
IF _w9 AND Liquidos.InyectarLiq[4] THEN Total := entradas.TR_L4_FT2_Tot.rtotal + AuxVol; END_IF
auxIniCal S= _w9 AND Modo_Calibrar_L4 OR _w9 AND Liquidos.InyectarLiq[4];

// NETWORK 27
_w10 := auxIniCal AND Modo_Calibrar_L4 AND entradas.CA1_L4_FT1_Tot.rtotal >= Total OR auxIniCal AND Liquidos.InyectarLiq[4] AND entradas.TR_L4_FT2_Tot.rtotal >= Total;
HMI.CA1_L4_V4_Cmd_Man R= _w10;
Liquidos.InyectarLiq[4] R= _w10;
Modo_Calibrar_L4 R= _w10;
auxIniCal R= _w10;
HMI.CmdM_PC1_L4_BD R= _w10;

// NETWORK 28
_w11 := Liquidos.InyectarLiq[4];
IF _w11 THEN Calculo_caudal_L4.Dosis := RECETA_ACTIVA.SetCircuitosLiq[4].Dosis; END_IF
IF _w11 THEN SetDemoraInyeccion := RECETA_ACTIVA.SetCircuitosLiq[4].Demora; END_IF
IF _w11 THEN Calculo_caudal_L4.TiempoInyeccion := RECETA_ACTIVA.SetCircuitosLiq[4].Inyeccion; END_IF
IF _w11 THEN Calculo_caudal_L4.Peso := Balanza_semilla.PesoSemilla_paraDosificar; END_IF

// NETWORK 29
_w12 := Modo_Calibrar_L4;
IF _w12 THEN Calculo_caudal_L4.Dosis := Puesto_CA1.CA1_Calibracion.Dosis; END_IF
IF _w12 THEN Calculo_caudal_L4.TiempoInyeccion := Puesto_CA1.CA1_Calibracion.TiempoIny; END_IF
IF _w12 THEN Calculo_caudal_L4.Peso := Puesto_CA1.CA1_Calibracion.PesoSemilla; END_IF

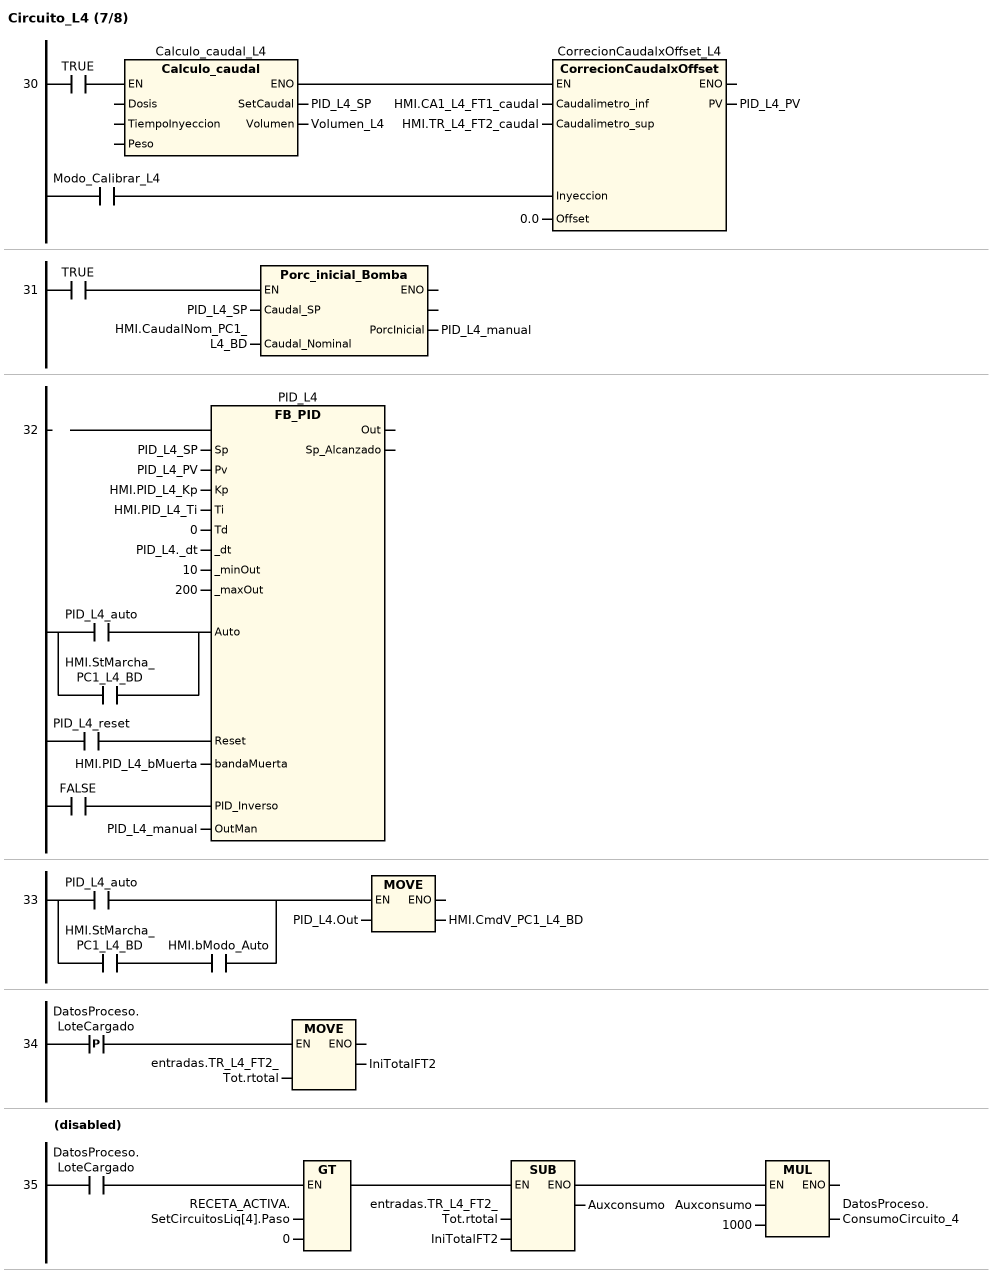
// NETWORK 30
Calculo_caudal_L4(SetCaudal => PID_L4_SP, Volumen => Volumen_L4); // Calculo_caudal
CorrecionCaudalxOffset_L4(
    Caudalimetro_inf := HMI.CA1_L4_FT1_caudal,
    Caudalimetro_sup := HMI.TR_L4_FT2_caudal,
    Inyeccion := Modo_Calibrar_L4,
    Offset := 0.0,
    PV => PID_L4_PV); // CorrecionCaudalxOffset

// NETWORK 31
Porc_inicial_Bomba(Caudal_SP := PID_L4_SP, Caudal_Nominal := HMI.CaudalNom_PC1_L4_BD, PorcInicial => PID_L4_manual);

// NETWORK 32
PID_L4(
    Sp := PID_L4_SP,
    Pv := PID_L4_PV,
    Kp := HMI.PID_L4_Kp,
    Ti := HMI.PID_L4_Ti,
    Td := 0,
    _dt := PID_L4._dt,
    _minOut := 10,
    _maxOut := 200,
    Auto := PID_L4_auto OR HMI.StMarcha_PC1_L4_BD,
    Reset := PID_L4_reset,
    bandaMuerta := HMI.PID_L4_bMuerta,
    PID_Inverso := FALSE,
    OutMan := PID_L4_manual); // FB_PID

// NETWORK 33
IF PID_L4_auto OR HMI.StMarcha_PC1_L4_BD AND HMI.bModo_Auto THEN HMI.CmdV_PC1_L4_BD := PID_L4.Out; END_IF

// NETWORK 34
_rt2(CLK := DatosProceso.LoteCargado);
IF _rt2.Q THEN IniTotalFT2 := entradas.TR_L4_FT2_Tot.rtotal; END_IF

// NETWORK 35 (disabled)
// _w13 := DatosProceso.LoteCargado AND RECETA_ACTIVA.SetCircuitosLiq[4].Paso > 0;
// IF _w13 THEN Auxconsumo := entradas.TR_L4_FT2_Tot.rtotal - IniTotalFT2; END_IF
// IF _w13 THEN DatosProceso.ConsumoCircuito_4 := Auxconsumo * 1000; END_IF

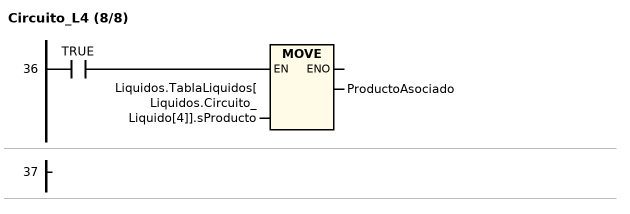
// NETWORK 36
ProductoAsociado := Liquidos.TablaLiquidos[Liquidos.Circuito_Liquido[4]].sProducto;

// NETWORK 37

END_PROGRAM

// ---- POUs/Puesto_Calibracion_2/Circuito_L5.TcPOU
PROGRAM Circuito_L5
VAR_INPUT
	Modo_Calibrar_L5: BOOL;
END_VAR
VAR
		fbBomba_L5 :Equipo_Motor_ATV320;
		ControlValv_ioLink_V1:ControlValv_ioLink;
		ControlValv_ioLink_V2: ControlValv_ioLink;
		ControlValv_ioLink_V3: ControlValv_ioLink;
		ControlValv_ioLink_V4: ControlValv_ioLink;
		Falla_L5_V1:BOOL;
		Falla_L5_V2:BOOL;
		Falla_L5_V3:BOOL;
		Falla_L5_V4:BOOL;
	Balanza_PU2_WT5: Balanza;
		dHS:DINT;
		TOF_calibradoIBC: TOF;
		PID_L5_SP:REAL;
		PID_L5_auto:BOOL;
		PID_L5_reset:BOOL;
		PID_L5_manual:REAL;
		PID_L5_bMuerta:REAL := 5;
		PID_L5_Kp:REAL := 0.1;
		PID_L5_Ti:REAL := 100;
		PID_L5_PV:REAL;
		Dosis_L5	:REAL;
		TiempoInyeccion_L5	:DINT;
		Peso	:REAL;
		Offset_L5:REAL;
		Inyeccion_L5:BOOL;

		Volumen_L5:REAL;
	Calculo_caudal_L5: Calculo_caudal;
	CorrecionCaudalxOffset_L5: CorrecionCaudalxOffset;
	tInyeccion: TON;
	Total :REAL;
	Totalant	:REAL;
	auxIniCal:BOOL;
	AuxVol5:REAL;
	TDemoraInyectar: TON;
	SetDemoraInyeccion: REAL;
	Tiempo_seg_to_TIME_DemoraInyec: Tiempo_seg_to_TIME;
	AuxTDemoraInyec: TIME;
	PID_L5: FB_PID;
	Tiempo_TIME_to_seg_InyCal: Tiempo_TIME_to_seg;
	AuxInyCal:TIME;
	ProductoAsociado: STRING;
	Lavagem_Circuito05: Lavagem;
	Teste: BOOL;
END_VAR

VAR PERSISTENT
	UltimaCalibracao	:UDINT;	//Data e hora da ultima calibração
END_VAR
VAR // added by the converter: edge detectors and wires of the graphical bodies
    _w1, _w2, _w3, _w4, _w5, _w6, _w7, _w8, _w9, _w10, _w11, _w12 : BOOL;
    _ft1 : F_TRIG;
    _rt1 : R_TRIG;
END_VAR

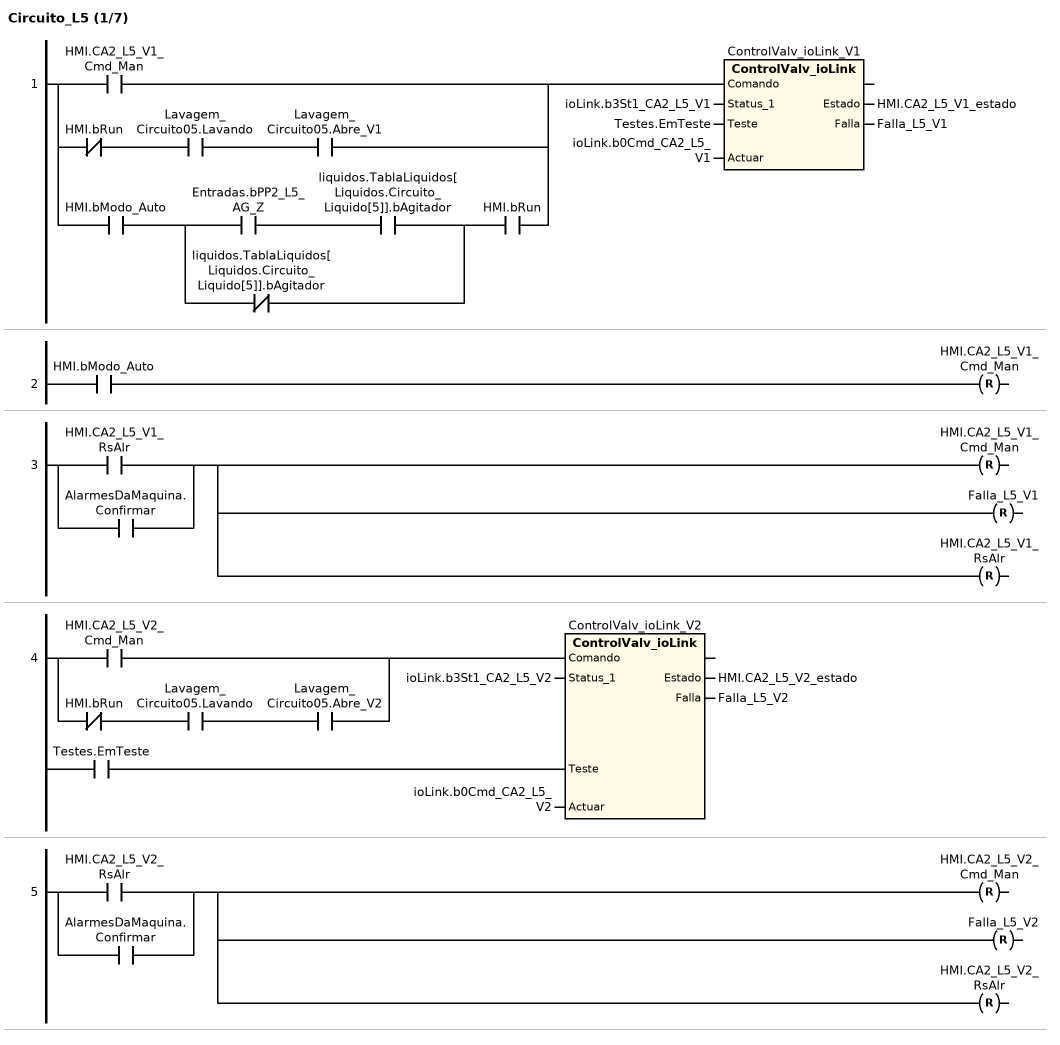
// NETWORK 1
ControlValv_ioLink_V1(
    Comando := HMI.CA2_L5_V1_Cmd_Man OR NOT HMI.bRun AND Lavagem_Circuito05.Lavando AND Lavagem_Circuito05.Abre_V1 OR HMI.bModo_Auto AND (Entradas.bPP2_L5_AG_Z AND (liquidos.TablaLiquidos[Liquidos.Circuito_Liquido[5]].bAgitador) OR NOT (liquidos.TablaLiquidos[Liquidos.Circuito_Liquido[5]].bAgitador)) AND HMI.bRun,
    Status_1 := ioLink.b3St1_CA2_L5_V1,
    Teste := Testes.EmTeste,
    Actuar := ioLink.b0Cmd_CA2_L5_V1,
    Estado => HMI.CA2_L5_V1_estado,
    Falla => Falla_L5_V1); // ControlValv_ioLink

// NETWORK 2
HMI.CA2_L5_V1_Cmd_Man R= HMI.bModo_Auto;

// NETWORK 3
_w1 := HMI.CA2_L5_V1_RsAlr OR AlarmesDaMaquina.Confirmar;
HMI.CA2_L5_V1_Cmd_Man R= _w1;
Falla_L5_V1 R= _w1;
HMI.CA2_L5_V1_RsAlr R= _w1;

// NETWORK 4
ControlValv_ioLink_V2(
    Comando := HMI.CA2_L5_V2_Cmd_Man OR NOT HMI.bRun AND Lavagem_Circuito05.Lavando AND Lavagem_Circuito05.Abre_V2,
    Status_1 := ioLink.b3St1_CA2_L5_V2,
    Teste := Testes.EmTeste,
    Actuar := ioLink.b0Cmd_CA2_L5_V2,
    Estado => HMI.CA2_L5_V2_estado,
    Falla => Falla_L5_V2); // ControlValv_ioLink

// NETWORK 5
_w2 := HMI.CA2_L5_V2_RsAlr OR AlarmesDaMaquina.Confirmar;
HMI.CA2_L5_V2_Cmd_Man R= _w2;
Falla_L5_V2 R= _w2;
HMI.CA2_L5_V2_RsAlr R= _w2;

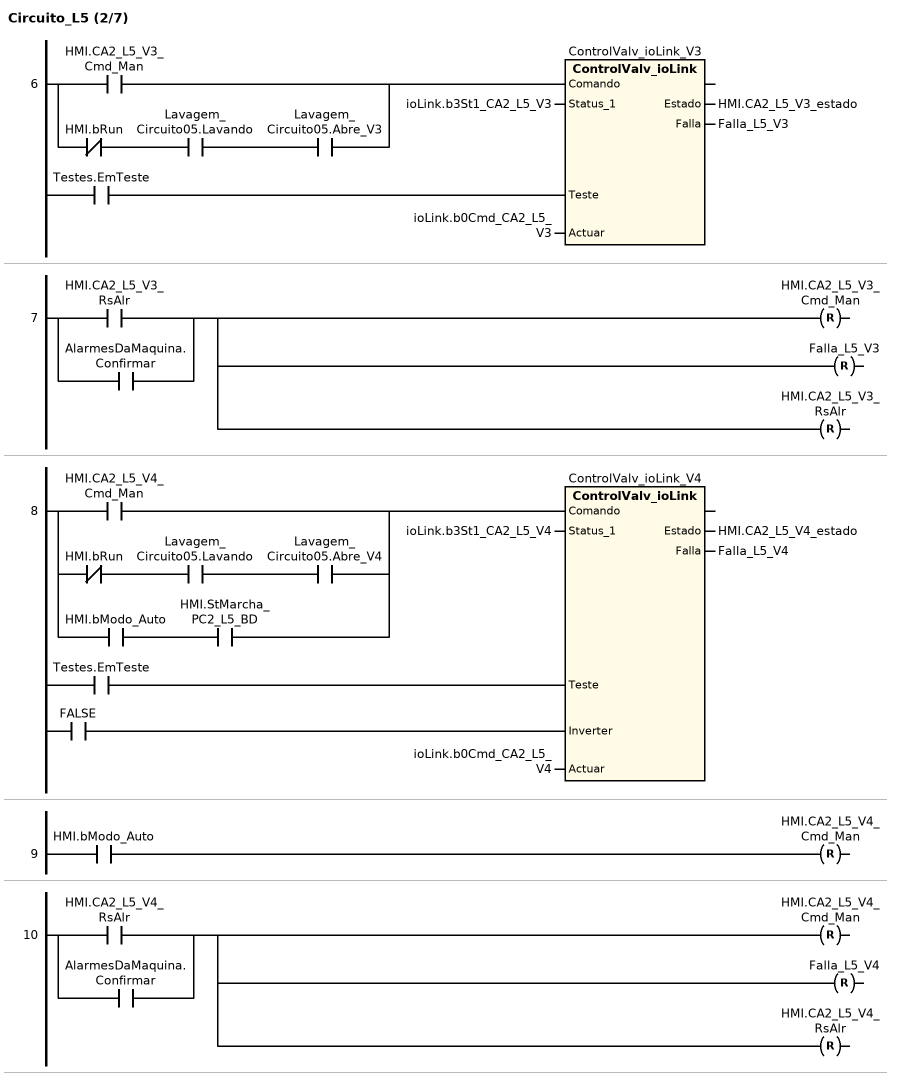
// NETWORK 6
ControlValv_ioLink_V3(
    Comando := HMI.CA2_L5_V3_Cmd_Man OR NOT HMI.bRun AND Lavagem_Circuito05.Lavando AND Lavagem_Circuito05.Abre_V3,
    Status_1 := ioLink.b3St1_CA2_L5_V3,
    Teste := Testes.EmTeste,
    Actuar := ioLink.b0Cmd_CA2_L5_V3,
    Estado => HMI.CA2_L5_V3_estado,
    Falla => Falla_L5_V3); // ControlValv_ioLink

// NETWORK 7
_w3 := HMI.CA2_L5_V3_RsAlr OR AlarmesDaMaquina.Confirmar;
HMI.CA2_L5_V3_Cmd_Man R= _w3;
Falla_L5_V3 R= _w3;
HMI.CA2_L5_V3_RsAlr R= _w3;

// NETWORK 8
ControlValv_ioLink_V4(
    Comando := HMI.CA2_L5_V4_Cmd_Man OR NOT HMI.bRun AND Lavagem_Circuito05.Lavando AND Lavagem_Circuito05.Abre_V4 OR HMI.bModo_Auto AND HMI.StMarcha_PC2_L5_BD,
    Status_1 := ioLink.b3St1_CA2_L5_V4,
    Teste := Testes.EmTeste,
    Inverter := FALSE,
    Actuar := ioLink.b0Cmd_CA2_L5_V4,
    Estado => HMI.CA2_L5_V4_estado,
    Falla => Falla_L5_V4); // ControlValv_ioLink

// NETWORK 9
HMI.CA2_L5_V4_Cmd_Man R= HMI.bModo_Auto;

// NETWORK 10
_w4 := HMI.CA2_L5_V4_RsAlr OR AlarmesDaMaquina.Confirmar;
HMI.CA2_L5_V4_Cmd_Man R= _w4;
Falla_L5_V4 R= _w4;
HMI.CA2_L5_V4_RsAlr R= _w4;

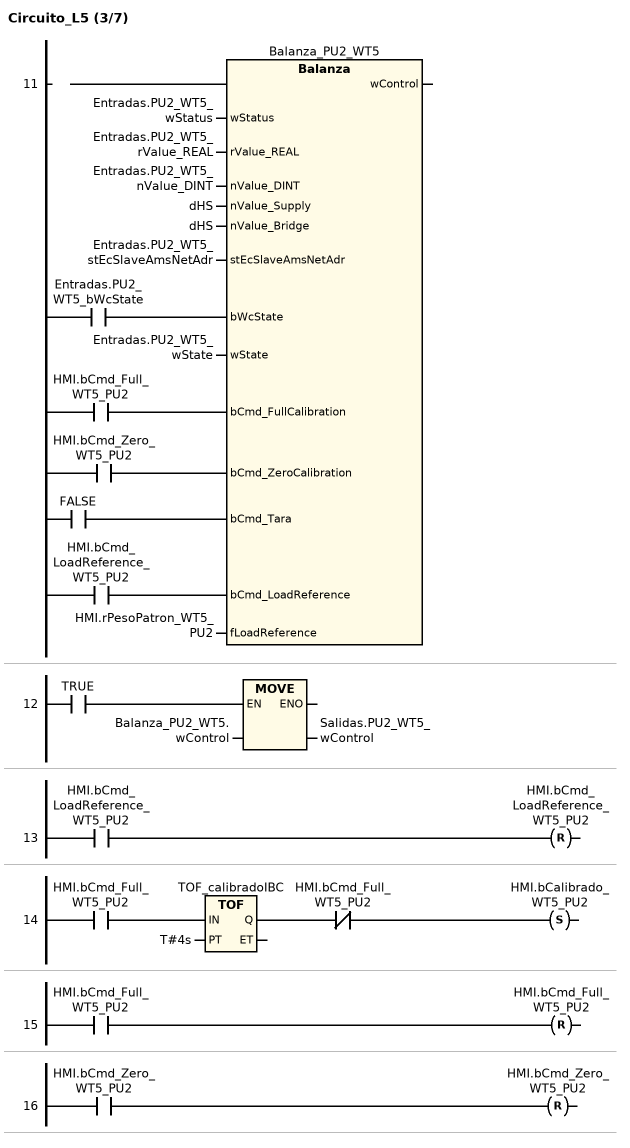
// NETWORK 11
Balanza_PU2_WT5(
    wStatus := Entradas.PU2_WT5_wStatus,
    rValue_REAL := Entradas.PU2_WT5_rValue_REAL,
    nValue_DINT := Entradas.PU2_WT5_nValue_DINT,
    nValue_Supply := dHS,
    nValue_Bridge := dHS,
    stEcSlaveAmsNetAdr := Entradas.PU2_WT5_stEcSlaveAmsNetAdr,
    bWcState := Entradas.PU2_WT5_bWcState,
    wState := Entradas.PU2_WT5_wState,
    bCmd_FullCalibration := HMI.bCmd_Full_WT5_PU2,
    bCmd_ZeroCalibration := HMI.bCmd_Zero_WT5_PU2,
    bCmd_Tara := FALSE,
    bCmd_LoadReference := HMI.bCmd_LoadReference_WT5_PU2,
    fLoadReference := HMI.rPesoPatron_WT5_PU2); // Balanza

// NETWORK 12
Salidas.PU2_WT5_wControl := Balanza_PU2_WT5.wControl;

// NETWORK 13
HMI.bCmd_LoadReference_WT5_PU2 R= HMI.bCmd_LoadReference_WT5_PU2;

// NETWORK 14
TOF_calibradoIBC(IN := HMI.bCmd_Full_WT5_PU2, PT := T#4s); // TOF
HMI.bCalibrado_WT5_PU2 S= TOF_calibradoIBC.Q AND NOT HMI.bCmd_Full_WT5_PU2;

// NETWORK 15
HMI.bCmd_Full_WT5_PU2 R= HMI.bCmd_Full_WT5_PU2;

// NETWORK 16
HMI.bCmd_Zero_WT5_PU2 R= HMI.bCmd_Zero_WT5_PU2;

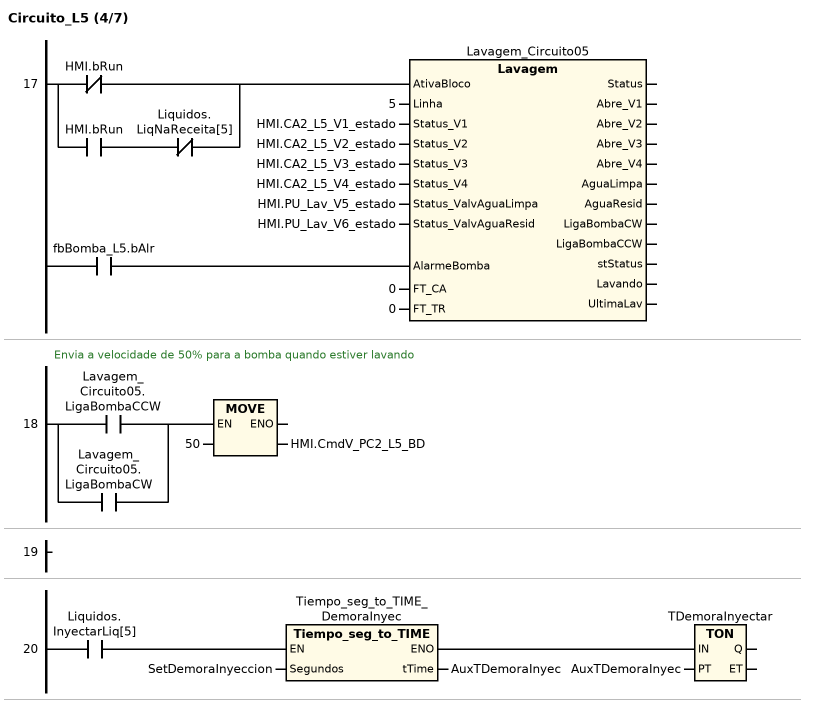
// NETWORK 17
Lavagem_Circuito05(
    AtivaBloco := NOT HMI.bRun OR HMI.bRun AND NOT Liquidos.LiqNaReceita[5],
    Linha := 5,
    Status_V1 := HMI.CA2_L5_V1_estado,
    Status_V2 := HMI.CA2_L5_V2_estado,
    Status_V3 := HMI.CA2_L5_V3_estado,
    Status_V4 := HMI.CA2_L5_V4_estado,
    Status_ValvAguaLimpa := HMI.PU_Lav_V5_estado,
    Status_ValvAguaResid := HMI.PU_Lav_V6_estado,
    AlarmeBomba := fbBomba_L5.bAlr,
    FT_CA := 0,
    FT_TR := 0); // Lavagem

// NETWORK 18
// Envia a velocidade de 50% para a bomba quando estiver lavando
IF Lavagem_Circuito05.LigaBombaCCW OR Lavagem_Circuito05.LigaBombaCW THEN HMI.CmdV_PC2_L5_BD := 50; END_IF

// NETWORK 19

// NETWORK 20
_w5 := Liquidos.InyectarLiq[5];
IF _w5 THEN
    Tiempo_seg_to_TIME_DemoraInyec(Segundos := SetDemoraInyeccion, tTime => AuxTDemoraInyec); // Tiempo_seg_to_TIME
END_IF
TDemoraInyectar(IN := _w5, PT := AuxTDemoraInyec); // TON

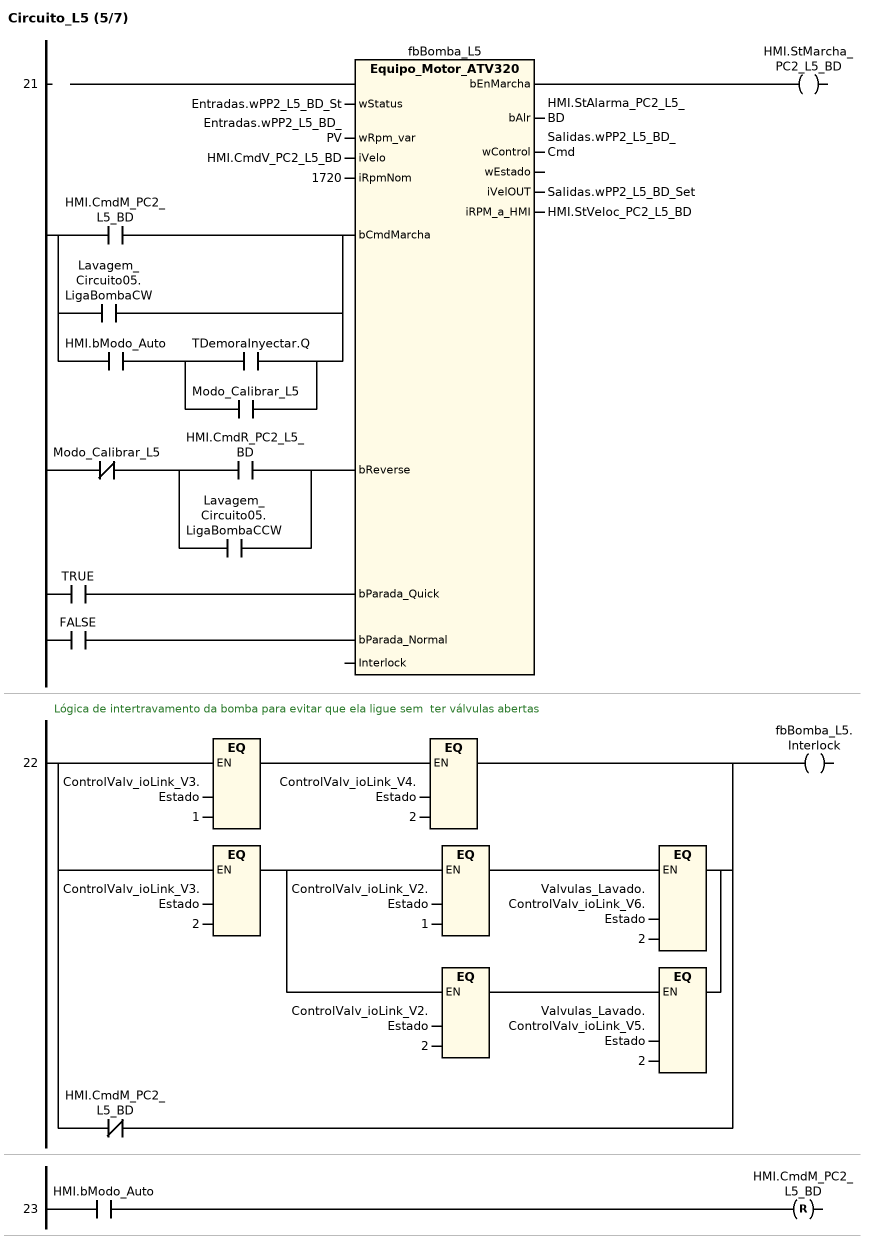
// NETWORK 21
fbBomba_L5(
    wStatus := Entradas.wPP2_L5_BD_St,
    wRpm_var := Entradas.wPP2_L5_BD_PV,
    iVelo := HMI.CmdV_PC2_L5_BD,
    iRpmNom := 1720,
    bCmdMarcha := HMI.CmdM_PC2_L5_BD OR Lavagem_Circuito05.LigaBombaCW OR HMI.bModo_Auto AND (TDemoraInyectar.Q OR Modo_Calibrar_L5),
    bReverse := NOT Modo_Calibrar_L5 AND (HMI.CmdR_PC2_L5_BD OR Lavagem_Circuito05.LigaBombaCCW),
    bParada_Quick := TRUE,
    bParada_Normal := FALSE,
    bAlr => HMI.StAlarma_PC2_L5_BD,
    wControl => Salidas.wPP2_L5_BD_Cmd,
    iVelOUT => Salidas.wPP2_L5_BD_Set,
    iRPM_a_HMI => HMI.StVeloc_PC2_L5_BD); // Equipo_Motor_ATV320
HMI.StMarcha_PC2_L5_BD := fbBomba_L5.bEnMarcha;

// NETWORK 22
// Lógica de intertravamento da bomba para evitar que ela ligue sem  ter válvulas abertas
_w6 := NOT HMI.CmdM_PC2_L5_BD;
IF NOT _w6 THEN
    _w7 := ControlValv_ioLink_V3.Estado = 2;
    _w6 := ControlValv_ioLink_V3.Estado = 1 AND ControlValv_ioLink_V4.Estado = 2 OR (_w7 AND ControlValv_ioLink_V2.Estado = 1 AND Valvulas_Lavado.ControlValv_ioLink_V6.Estado = 2 OR _w7 AND ControlValv_ioLink_V2.Estado = 2 AND Valvulas_Lavado.ControlValv_ioLink_V5.Estado = 2);
END_IF
fbBomba_L5.Interlock := _w6;

// NETWORK 23
HMI.CmdM_PC2_L5_BD R= HMI.bModo_Auto;

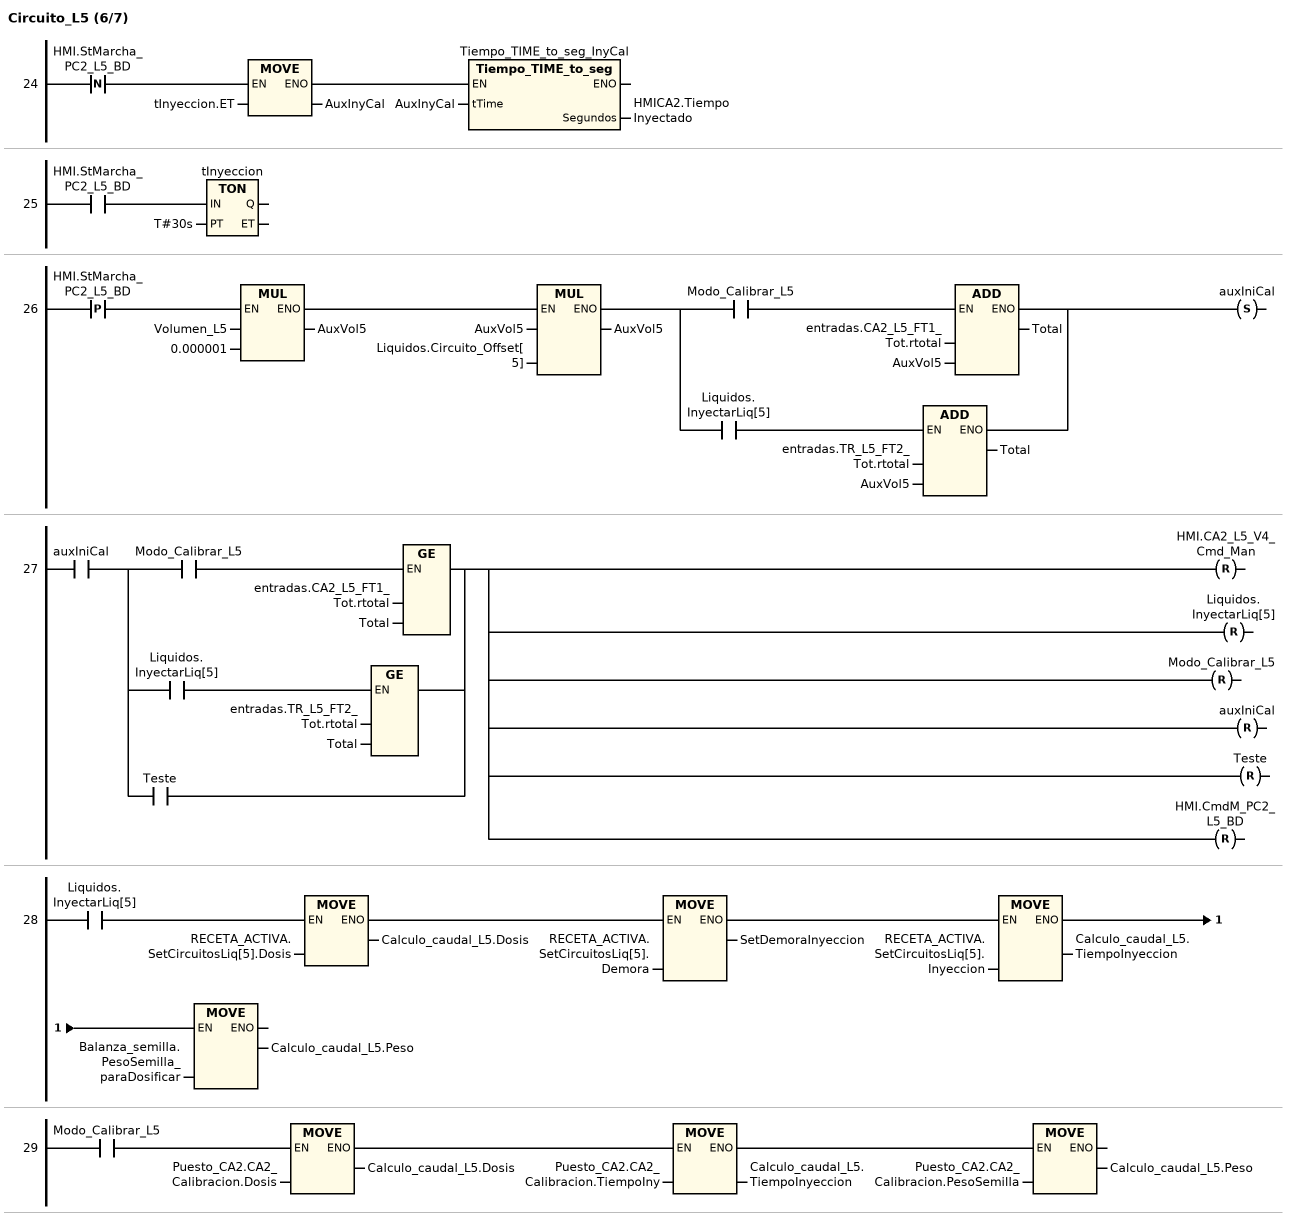
// NETWORK 24
_ft1(CLK := HMI.StMarcha_PC2_L5_BD);
_w8 := _ft1.Q;
IF _w8 THEN AuxInyCal := tInyeccion.ET; END_IF
IF _w8 THEN
    Tiempo_TIME_to_seg_InyCal(tTime := AuxInyCal, Segundos => HMICA2.TiempoInyectado); // Tiempo_TIME_to_seg
END_IF

// NETWORK 25
tInyeccion(IN := HMI.StMarcha_PC2_L5_BD, PT := T#30s); // TON

// NETWORK 26
_rt1(CLK := HMI.StMarcha_PC2_L5_BD);
_w9 := _rt1.Q;
IF _w9 THEN AuxVol5 := Volumen_L5 * 0.000001; END_IF
IF _w9 THEN AuxVol5 := AuxVol5 * Liquidos.Circuito_Offset[5]; END_IF
IF _w9 AND Modo_Calibrar_L5 THEN Total := entradas.CA2_L5_FT1_Tot.rtotal + AuxVol5; END_IF
IF _w9 AND Liquidos.InyectarLiq[5] THEN Total := entradas.TR_L5_FT2_Tot.rtotal + AuxVol5; END_IF
auxIniCal S= _w9 AND Modo_Calibrar_L5 OR _w9 AND Liquidos.InyectarLiq[5];

// NETWORK 27
_w10 := auxIniCal AND Modo_Calibrar_L5 AND entradas.CA2_L5_FT1_Tot.rtotal >= Total OR (auxIniCal AND Liquidos.InyectarLiq[5] AND entradas.TR_L5_FT2_Tot.rtotal >= Total OR auxIniCal AND Teste);
HMI.CA2_L5_V4_Cmd_Man R= _w10;
Liquidos.InyectarLiq[5] R= _w10;
Modo_Calibrar_L5 R= _w10;
auxIniCal R= _w10;
Teste R= _w10;
HMI.CmdM_PC2_L5_BD R= _w10;

// NETWORK 28
_w11 := Liquidos.InyectarLiq[5];
IF _w11 THEN Calculo_caudal_L5.Dosis := RECETA_ACTIVA.SetCircuitosLiq[5].Dosis; END_IF
IF _w11 THEN SetDemoraInyeccion := RECETA_ACTIVA.SetCircuitosLiq[5].Demora; END_IF
IF _w11 THEN Calculo_caudal_L5.TiempoInyeccion := RECETA_ACTIVA.SetCircuitosLiq[5].Inyeccion; END_IF
IF _w11 THEN Calculo_caudal_L5.Peso := Balanza_semilla.PesoSemilla_paraDosificar; END_IF

// NETWORK 29
_w12 := Modo_Calibrar_L5;
IF _w12 THEN Calculo_caudal_L5.Dosis := Puesto_CA2.CA2_Calibracion.Dosis; END_IF
IF _w12 THEN Calculo_caudal_L5.TiempoInyeccion := Puesto_CA2.CA2_Calibracion.TiempoIny; END_IF
IF _w12 THEN Calculo_caudal_L5.Peso := Puesto_CA2.CA2_Calibracion.PesoSemilla; END_IF

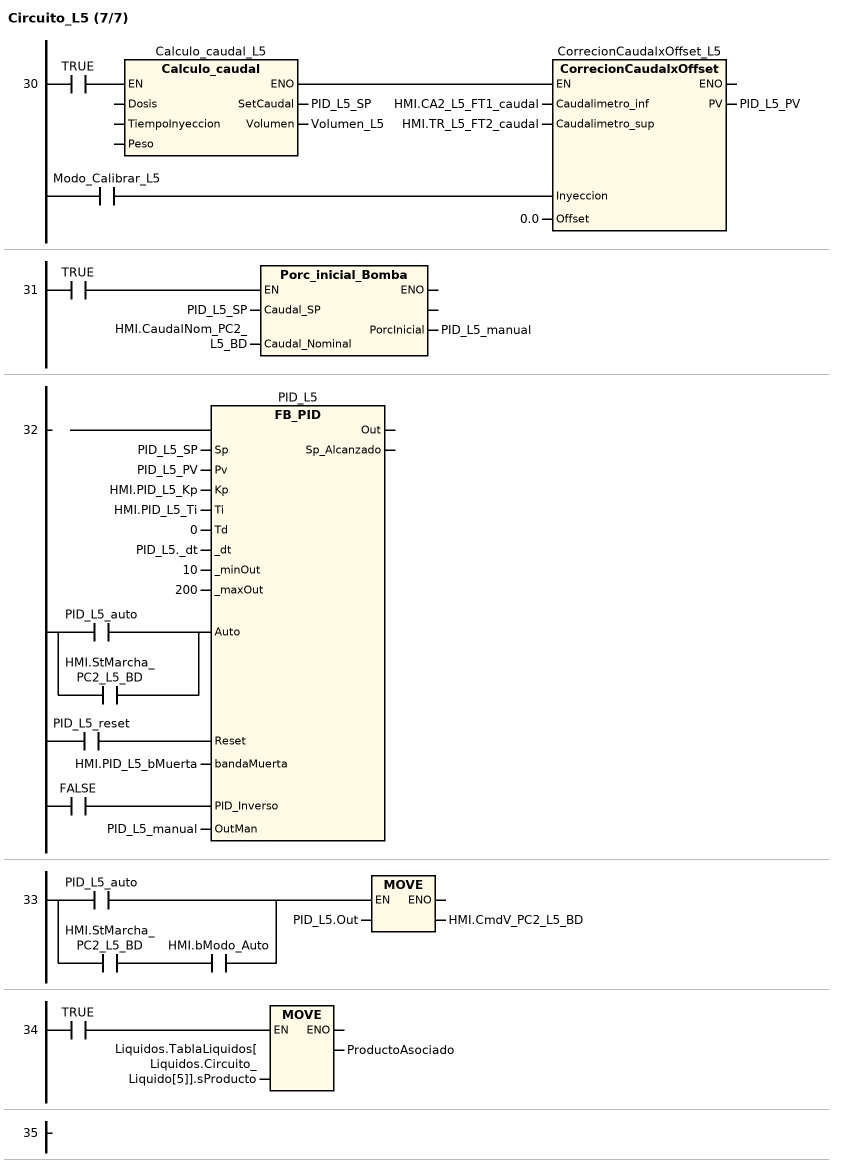
// NETWORK 30
Calculo_caudal_L5(SetCaudal => PID_L5_SP, Volumen => Volumen_L5); // Calculo_caudal
CorrecionCaudalxOffset_L5(
    Caudalimetro_inf := HMI.CA2_L5_FT1_caudal,
    Caudalimetro_sup := HMI.TR_L5_FT2_caudal,
    Inyeccion := Modo_Calibrar_L5,
    Offset := 0.0,
    PV => PID_L5_PV); // CorrecionCaudalxOffset

// NETWORK 31
Porc_inicial_Bomba(Caudal_SP := PID_L5_SP, Caudal_Nominal := HMI.CaudalNom_PC2_L5_BD, PorcInicial => PID_L5_manual);

// NETWORK 32
PID_L5(
    Sp := PID_L5_SP,
    Pv := PID_L5_PV,
    Kp := HMI.PID_L5_Kp,
    Ti := HMI.PID_L5_Ti,
    Td := 0,
    _dt := PID_L5._dt,
    _minOut := 10,
    _maxOut := 200,
    Auto := PID_L5_auto OR HMI.StMarcha_PC2_L5_BD,
    Reset := PID_L5_reset,
    bandaMuerta := HMI.PID_L5_bMuerta,
    PID_Inverso := FALSE,
    OutMan := PID_L5_manual); // FB_PID

// NETWORK 33
IF PID_L5_auto OR HMI.StMarcha_PC2_L5_BD AND HMI.bModo_Auto THEN HMI.CmdV_PC2_L5_BD := PID_L5.Out; END_IF

// NETWORK 34
ProductoAsociado := Liquidos.TablaLiquidos[Liquidos.Circuito_Liquido[5]].sProducto;

// NETWORK 35

END_PROGRAM

// ---- POUs/Puesto_Calibracion_2/Puesto_CA2.TcPOU
PROGRAM Puesto_CA2
VAR
	Balanza_CA2: Balanza;
	dHS:DINT;
	Cmd_Full: R_TRIG;
	TmrLabelFinalizado: TON;
	AuxFinCalibrar:BOOL;
	CA2_Calibracion: Calibracion_Liq_calc;
	Tarar_balanza :BOOL;
	Offset_ref2:REAL;
	Inyectar_ref2:BOOL;
	InicioCal_ref2:BOOL;
	Offset_ref: REAL;
	Inyectar_ref: BOOL;
	InicioCal_ref: BOOL;

	UltimaCalibracao: UDINT;
	VazaoMax: REAL;
	VazaoMaxExcedida: BOOL;
END_VAR

//Indica a ultima calibração da linha selecionada
UltimaCalibracao := HMI.UltimasCalibracoes[HMI.iCircuito_a_calibrar];


Balanza_CA2(
	wStatus:=Entradas.CA2_WT1_wStatus , 
	rValue_REAL:=Entradas.CA2_WT1_rValue_REAL , 
	nValue_DINT:=Entradas.CA2_WT1_nValue_DINT , 
	nValue_Supply:=dHS , 
	nValue_Bridge:=dHS , 
	stEcSlaveAmsNetAdr:=Entradas.CA2_WT1_stEcSlaveAmsNetAdr , 
	bWcState:=Entradas.CA2_WT1_bWcState , 
	wState:=Entradas.CA2_WT1_wState , 
	bCmd_FullCalibration:=HMI.bCmd_Full_WT_CA2 , 
	bCmd_ZeroCalibration:=HMI.bCmd_Zero_WT_CA2 , 
	bCmd_Tara:=Tarar_balanza , 
	bCmd_LoadReference:=HMI.bCmd_LoadReference_WT_CA2 ,
	fLoadReference:=(HMI.rPesoPatron_WT_CA2)/1000,
	wControl=>Salidas.CA2_WT1_wControl );
	
	TmrLabelFinalizado(IN:= HMI.bCmd_Full_WT_CA2 , PT:=T#10S , Q=> , ET=> );
	
	HMI.bCmd_LoadReference_WT_CA2:=FALSE;
	HMI.bCmd_Zero_WT_CA2:=FALSE;
	HMI.bCmd_Full_WT_CA2:=FALSE;
	Tarar_balanza:=FALSE;
	Cmd_Full(CLK:=TmrLabelFinalizado.Q , Q=> );
	IF 	Cmd_Full.Q THEN
		HMI.bCalibrado_WT_CA2:=TRUE;
	END_IF
/////////////////
IF (4<HMI.iCircuito_a_calibrar AND HMI.iCircuito_a_calibrar<9) THEN
//
/////////
CASE HMI.iCircuito_a_calibrar OF
	5:	Offset_ref:=Liquidos.Circuito_Offset[5];
		Inyectar_ref:=circuito_L5.Modo_Calibrar_L5;
		InicioCal_ref:=HMICA2.Inicio_calibracion;
		HMICA2.VolumenPedido_calibracion:=circuito_L5.Volumen_L5;
	6:	Offset_ref:=Liquidos.Circuito_Offset[6];
		Inyectar_ref:=circuito_L6.Modo_Calibrar_L6;
		InicioCal_ref:=HMICA2.Inicio_calibracion;
		HMICA2.VolumenPedido_calibracion:=circuito_L6.Volumen_L6;
	7:	Offset_ref:=Liquidos.Circuito_Offset[7];
		Inyectar_ref:=circuito_L7.Modo_Calibrar_L7;
		InicioCal_ref:=HMICA2.Inicio_calibracion;
		HMICA2.VolumenPedido_calibracion:=circuito_L7.Volumen_L7;
	8:	Offset_ref:=Liquidos.Circuito_Offset[8];
		Inyectar_ref:=circuito_L8.Modo_Calibrar_L8;
		InicioCal_ref:=HMICA2.Inicio_calibracion;
		HMICA2.VolumenPedido_calibracion:=circuito_L8.Volumen_L8;	
		
		ELSE
	;		
END_CASE
CA2_Calibracion(
	Dosis:=HMICA2.Dosis_calibracion , 
	PesoSemilla:=HMICA2.Peso_calibracion,
	Tolerancia:=HMICA2.Tolerancia_calibracion , 
	PesoBalanza:=Entradas.CA2_WT1_rValue_REAL ,
	mlPedido:= HMICA2.VolumenPedido_calibracion,
	PesoEspec:=Puesto_CA1.PesoEspec , 
	Offset:=Offset_ref ,
	TiempoIny:=HMICA2.TInyeccion_calibracion , 
	Vol_Probeta:=(HMICA2.VolMaxProbeta_calibracion*1000) , 
	Pausa:=HMICA2.Pausa_calibracion , 
	Dosificar=> , 
	Probeta_Llena:=HMICA2.VaciarProbeta_calibracion , 
	Inyectar:=Inyectar_ref, 
	ml:=HMICA2.Volumen_calibracion, 
	Tiempo:=HMICA2.Tiempo_calibracion , 
	InicioCal:= InicioCal_ref, 
	Continuar:=HMICA2.Continuar_calibracion , 
	Tarar:=Tarar_balanza,
	Finalizado:=HMICA2.Fin_calibracion,
	mlProbeta=>HMICA2.Vol_enProbeta , 
	TiempoInyectado:=HMICA2.TiempoInyectado,
	Error_promedio=> HMICA2.Error_promedio, );
//
CASE HMI.iCircuito_a_calibrar OF
	5:	Liquidos.Circuito_Offset[5]:=Offset_ref;//Offset_ref
		circuito_L5.Modo_Calibrar_L5:=Inyectar_ref;//Inyectar_ref
		HMICA2.Inicio_calibracion:=InicioCal_ref;
		VazaoMax := HMI.CaudalNom_PC2_L5_BD;
	6:	Liquidos.Circuito_Offset[6]:=Offset_ref;//Offset_ref
		circuito_L6.Modo_Calibrar_L6:=Inyectar_ref;//Inyectar_ref
		HMICA2.Inicio_calibracion:=InicioCal_ref;
		VazaoMax := HMI.CaudalNom_PC2_L6_BD;
	7:	Liquidos.Circuito_Offset[7]:=Offset_ref;//Offset_ref
		circuito_L7.Modo_Calibrar_L7:=Inyectar_ref;//Inyectar_ref
		HMICA2.Inicio_calibracion:=InicioCal_ref;
		VazaoMax := HMI.CaudalNom_PC2_L7_BD;
	8:	Liquidos.Circuito_Offset[8]:=Offset_ref;//Offset_ref
		circuito_L8.Modo_Calibrar_L8:=Inyectar_ref;//Inyectar_ref
		HMICA2.Inicio_calibracion:=InicioCal_ref;
		VazaoMax := HMI.CaudalNom_PC2_L8_BD;
		
		ELSE
	;		
END_CASE	
END_IF	

IF HMICA2.TInyeccion_calibracion > 0 THEN
	IF (HMICA2.Dosis_calibracion*HMICA2.Peso_calibracion/100)/TO_REAL(HMICA2.TInyeccion_calibracion) > VazaoMax THEN
		VazaoMaxExcedida := TRUE;
	ELSE
		VazaoMaxExcedida := FALSE;
	END_IF
END_IF

END_PROGRAM

// ---- POUs/Puesto_Calibracion_2/Circuito_L6.TcPOU
PROGRAM Circuito_L6
VAR_INPUT
	Modo_Calibrar_L6: BOOL;
END_VAR
VAR
		fbBomba_L6 :Equipo_Motor_ATV320;
		ControlValv_ioLink_V1:ControlValv_ioLink;
		ControlValv_ioLink_V2: ControlValv_ioLink;
		ControlValv_ioLink_V3: ControlValv_ioLink;
		ControlValv_ioLink_V4: ControlValv_ioLink;
		Falla_L6_V1:BOOL;
		Falla_L6_V2:BOOL;
		Falla_L6_V3:BOOL;
		Falla_L6_V4:BOOL;
		Balanza_PU2_WT6: Balanza;
		dHS:DINT;
		TOF_calibradoIBC: TOF;
		PID_L6_SP		:REAL;
		PID_L6_auto		:BOOL;
		PID_L6_reset	:BOOL;
		PID_L6_manual	:REAL;
		PID_L6_bMuerta	:REAL := 5;
		PID_L6_Kp		:REAL := 0.1;
		PID_L6_Ti		:REAL := 100;
		PID_L6_PV		:REAL;
		Dosis_L6		:REAL;
		TiempoInyeccion_L6	:DINT;
		Peso	:REAL;
		Offset_L6:REAL;
		Inyeccion_L6:BOOL;
		Volumen_L6:REAL;
		Calculo_caudal_L6: Calculo_caudal;
		CorrecionCaudalxOffset_L6: CorrecionCaudalxOffset;
		tInyeccion: TON;
		Total :REAL;
		Totalant	:REAL;
		auxIniCal:BOOL;
		AuxVol:REAL;
		CA2_L6_V1_CmdA_Man :BOOL;
		CA2_L6_V4_CmdA_Man :BOOL;
		TDemoraInyectar: TON;
		SetDemoraInyeccion: REAL;
		Tiempo_seg_to_TIME_DemoraInyec: Tiempo_seg_to_TIME;
		AuxTDemoraInyec: TIME;
		PID_L6: FB_PID;	
		Tiempo_TIME_to_seg_InyCal: Tiempo_TIME_to_seg;
		AuxInyCal:TIME;	
	ProductoAsociado: STRING;
	Lavagem_Circuito06: Lavagem;
	Filtro2_0: Filtro2;
END_VAR

VAR PERSISTENT
	UltimaCalibracao	:UDINT;	//Data e hora da ultima calibração
END_VAR
VAR // added by the converter: edge detectors and wires of the graphical bodies
    _w1, _w2, _w3, _w4, _w5, _w6, _w7, _w8, _w9, _w10, _w11, _w12 : BOOL;
    _ft1 : F_TRIG;
    _rt1 : R_TRIG;
END_VAR

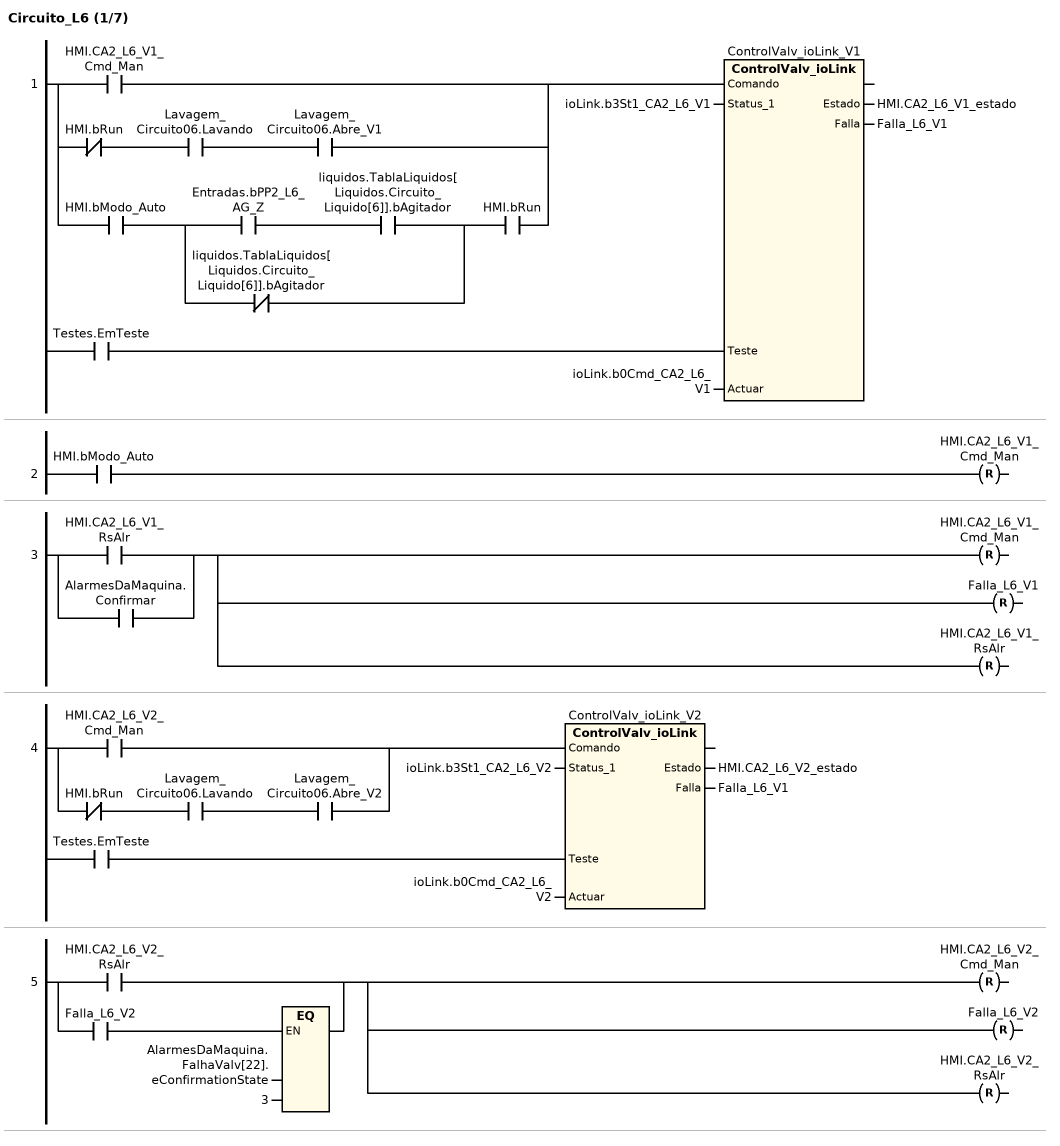
// NETWORK 1
ControlValv_ioLink_V1(
    Comando := HMI.CA2_L6_V1_Cmd_Man OR NOT HMI.bRun AND Lavagem_Circuito06.Lavando AND Lavagem_Circuito06.Abre_V1 OR HMI.bModo_Auto AND (Entradas.bPP2_L6_AG_Z AND (liquidos.TablaLiquidos[Liquidos.Circuito_Liquido[6]].bAgitador) OR NOT (liquidos.TablaLiquidos[Liquidos.Circuito_Liquido[6]].bAgitador)) AND HMI.bRun,
    Status_1 := ioLink.b3St1_CA2_L6_V1,
    Teste := Testes.EmTeste,
    Actuar := ioLink.b0Cmd_CA2_L6_V1,
    Estado => HMI.CA2_L6_V1_estado,
    Falla => Falla_L6_V1); // ControlValv_ioLink

// NETWORK 2
HMI.CA2_L6_V1_Cmd_Man R= HMI.bModo_Auto;

// NETWORK 3
_w1 := HMI.CA2_L6_V1_RsAlr OR AlarmesDaMaquina.Confirmar;
HMI.CA2_L6_V1_Cmd_Man R= _w1;
Falla_L6_V1 R= _w1;
HMI.CA2_L6_V1_RsAlr R= _w1;

// NETWORK 4
ControlValv_ioLink_V2(
    Comando := HMI.CA2_L6_V2_Cmd_Man OR NOT HMI.bRun AND Lavagem_Circuito06.Lavando AND Lavagem_Circuito06.Abre_V2,
    Status_1 := ioLink.b3St1_CA2_L6_V2,
    Teste := Testes.EmTeste,
    Actuar := ioLink.b0Cmd_CA2_L6_V2,
    Estado => HMI.CA2_L6_V2_estado,
    Falla => Falla_L6_V1); // ControlValv_ioLink

// NETWORK 5
_w2 := HMI.CA2_L6_V2_RsAlr OR Falla_L6_V2 AND AlarmesDaMaquina.FalhaValv[22].eConfirmationState = 3;
HMI.CA2_L6_V2_Cmd_Man R= _w2;
Falla_L6_V2 R= _w2;
HMI.CA2_L6_V2_RsAlr R= _w2;

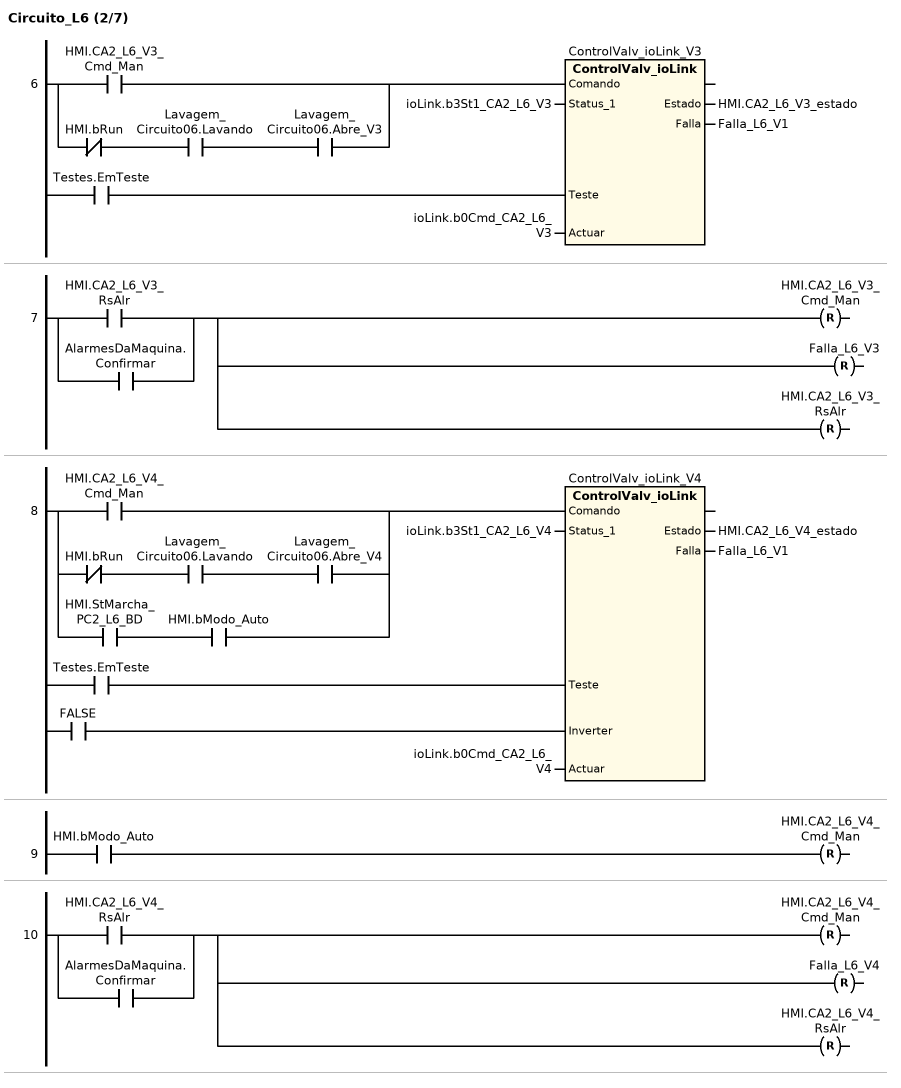
// NETWORK 6
ControlValv_ioLink_V3(
    Comando := HMI.CA2_L6_V3_Cmd_Man OR NOT HMI.bRun AND Lavagem_Circuito06.Lavando AND Lavagem_Circuito06.Abre_V3,
    Status_1 := ioLink.b3St1_CA2_L6_V3,
    Teste := Testes.EmTeste,
    Actuar := ioLink.b0Cmd_CA2_L6_V3,
    Estado => HMI.CA2_L6_V3_estado,
    Falla => Falla_L6_V1); // ControlValv_ioLink

// NETWORK 7
_w3 := HMI.CA2_L6_V3_RsAlr OR AlarmesDaMaquina.Confirmar;
HMI.CA2_L6_V3_Cmd_Man R= _w3;
Falla_L6_V3 R= _w3;
HMI.CA2_L6_V3_RsAlr R= _w3;

// NETWORK 8
ControlValv_ioLink_V4(
    Comando := HMI.CA2_L6_V4_Cmd_Man OR NOT HMI.bRun AND Lavagem_Circuito06.Lavando AND Lavagem_Circuito06.Abre_V4 OR HMI.StMarcha_PC2_L6_BD AND HMI.bModo_Auto,
    Status_1 := ioLink.b3St1_CA2_L6_V4,
    Teste := Testes.EmTeste,
    Inverter := FALSE,
    Actuar := ioLink.b0Cmd_CA2_L6_V4,
    Estado => HMI.CA2_L6_V4_estado,
    Falla => Falla_L6_V1); // ControlValv_ioLink

// NETWORK 9
HMI.CA2_L6_V4_Cmd_Man R= HMI.bModo_Auto;

// NETWORK 10
_w4 := HMI.CA2_L6_V4_RsAlr OR AlarmesDaMaquina.Confirmar;
HMI.CA2_L6_V4_Cmd_Man R= _w4;
Falla_L6_V4 R= _w4;
HMI.CA2_L6_V4_RsAlr R= _w4;

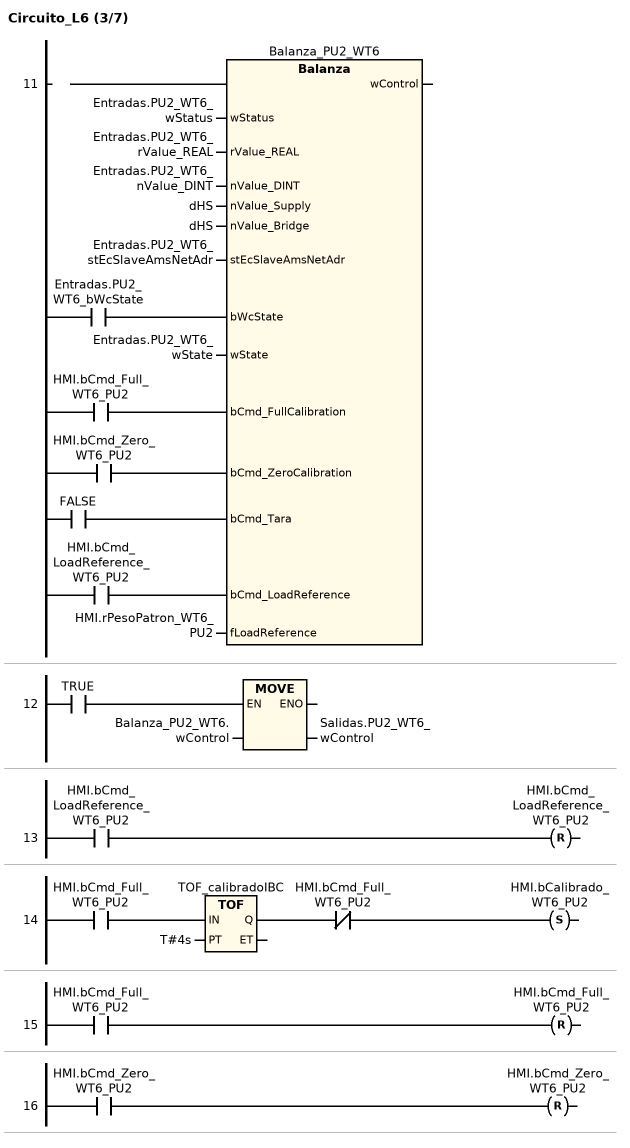
// NETWORK 11
Balanza_PU2_WT6(
    wStatus := Entradas.PU2_WT6_wStatus,
    rValue_REAL := Entradas.PU2_WT6_rValue_REAL,
    nValue_DINT := Entradas.PU2_WT6_nValue_DINT,
    nValue_Supply := dHS,
    nValue_Bridge := dHS,
    stEcSlaveAmsNetAdr := Entradas.PU2_WT6_stEcSlaveAmsNetAdr,
    bWcState := Entradas.PU2_WT6_bWcState,
    wState := Entradas.PU2_WT6_wState,
    bCmd_FullCalibration := HMI.bCmd_Full_WT6_PU2,
    bCmd_ZeroCalibration := HMI.bCmd_Zero_WT6_PU2,
    bCmd_Tara := FALSE,
    bCmd_LoadReference := HMI.bCmd_LoadReference_WT6_PU2,
    fLoadReference := HMI.rPesoPatron_WT6_PU2); // Balanza

// NETWORK 12
Salidas.PU2_WT6_wControl := Balanza_PU2_WT6.wControl;

// NETWORK 13
HMI.bCmd_LoadReference_WT6_PU2 R= HMI.bCmd_LoadReference_WT6_PU2;

// NETWORK 14
TOF_calibradoIBC(IN := HMI.bCmd_Full_WT6_PU2, PT := T#4s); // TOF
HMI.bCalibrado_WT6_PU2 S= TOF_calibradoIBC.Q AND NOT HMI.bCmd_Full_WT6_PU2;

// NETWORK 15
HMI.bCmd_Full_WT6_PU2 R= HMI.bCmd_Full_WT6_PU2;

// NETWORK 16
HMI.bCmd_Zero_WT6_PU2 R= HMI.bCmd_Zero_WT6_PU2;

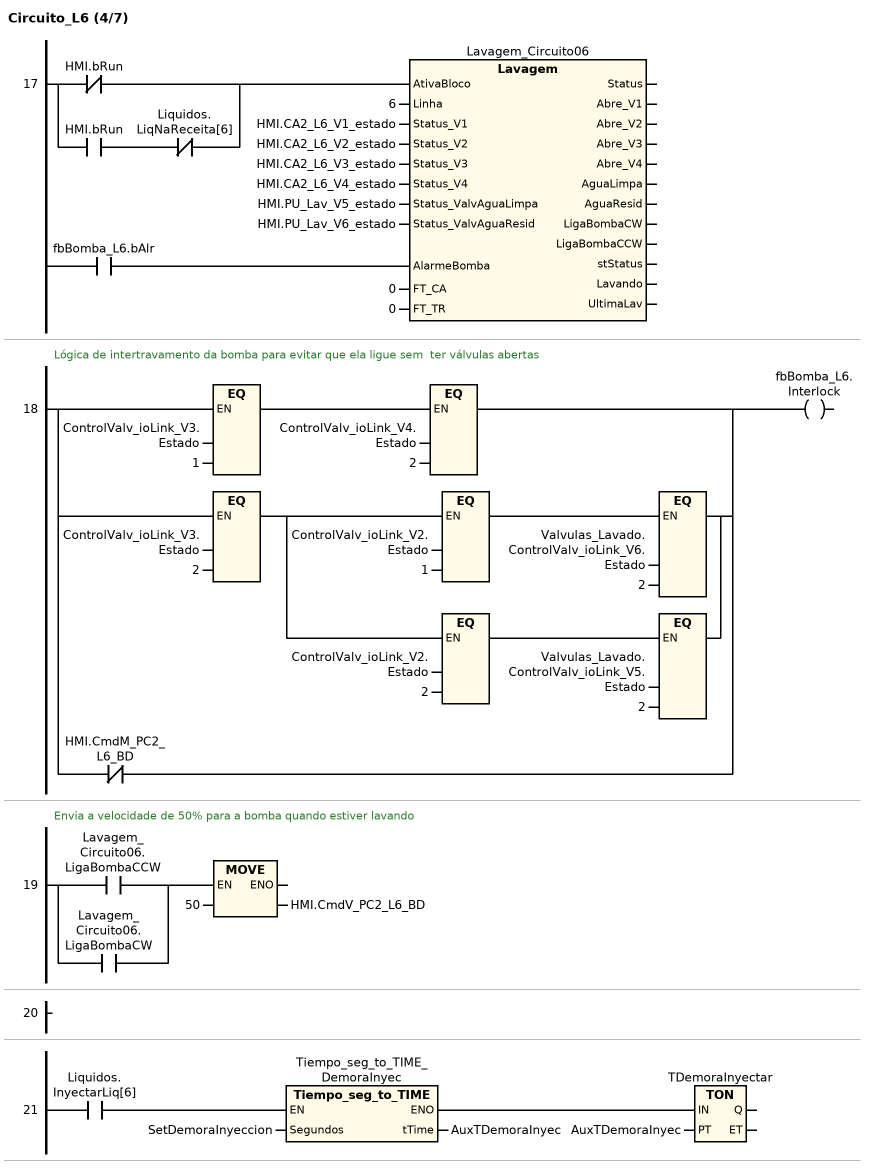
// NETWORK 17
Lavagem_Circuito06(
    AtivaBloco := NOT HMI.bRun OR HMI.bRun AND NOT Liquidos.LiqNaReceita[6],
    Linha := 6,
    Status_V1 := HMI.CA2_L6_V1_estado,
    Status_V2 := HMI.CA2_L6_V2_estado,
    Status_V3 := HMI.CA2_L6_V3_estado,
    Status_V4 := HMI.CA2_L6_V4_estado,
    Status_ValvAguaLimpa := HMI.PU_Lav_V5_estado,
    Status_ValvAguaResid := HMI.PU_Lav_V6_estado,
    AlarmeBomba := fbBomba_L6.bAlr,
    FT_CA := 0,
    FT_TR := 0); // Lavagem

// NETWORK 18
// Lógica de intertravamento da bomba para evitar que ela ligue sem  ter válvulas abertas
_w5 := NOT HMI.CmdM_PC2_L6_BD;
IF NOT _w5 THEN
    _w6 := ControlValv_ioLink_V3.Estado = 2;
    _w5 := ControlValv_ioLink_V3.Estado = 1 AND ControlValv_ioLink_V4.Estado = 2 OR (_w6 AND ControlValv_ioLink_V2.Estado = 1 AND Valvulas_Lavado.ControlValv_ioLink_V6.Estado = 2 OR _w6 AND ControlValv_ioLink_V2.Estado = 2 AND Valvulas_Lavado.ControlValv_ioLink_V5.Estado = 2);
END_IF
fbBomba_L6.Interlock := _w5;

// NETWORK 19
// Envia a velocidade de 50% para a bomba quando estiver lavando
IF Lavagem_Circuito06.LigaBombaCCW OR Lavagem_Circuito06.LigaBombaCW THEN HMI.CmdV_PC2_L6_BD := 50; END_IF

// NETWORK 20

// NETWORK 21
_w7 := Liquidos.InyectarLiq[6];
IF _w7 THEN
    Tiempo_seg_to_TIME_DemoraInyec(Segundos := SetDemoraInyeccion, tTime => AuxTDemoraInyec); // Tiempo_seg_to_TIME
END_IF
TDemoraInyectar(IN := _w7, PT := AuxTDemoraInyec); // TON

